LIN {X 0,Y 446.455,Z 877.557,A -85,B 0,C 180,E1 -8817.293,E2 -8817.293} C_VEL
LIN {X 0,Y 446.313,Z 878.965,A -85,B 0,C 180,E1 -8819.098,E2 -8819.098} C_VEL
LIN {X 0,Y 446.282,Z 879.074,A -85,B 0,C 180,E1 -8820,E2 -8820} C_VEL
LIN {X 0,Y 446.28,Z 878.729,A -85,B 0,C 180,E1 -8820.902,E2 -8820.902} C_VEL
LIN {X 0,Y 446.154,Z 876.876,A -85,B 0,C 180,E1 -8822.709,E2 -8822.709} C_VEL
LIN {X 0,Y 446.322,Z 874.333,A -85,B 0,C 180,E1 -8824.063,E2 -8824.063} C_VEL
LIN {X 0,Y 446.471,Z 870.782,A -85,B 0,C 180,E1 -8825.42,E2 -8825.42} C_VEL
LIN {X 0,Y 446.753,Z 866.002,A -85,B 0,C 180,E1 -8826.798,E2 -8826.798} C_VEL
LIN {X 0,Y 446.982,Z 860.13,A -85,B 0,C 180,E1 -8828.135,E2 -8828.135} C_VEL
LIN {X 0,Y 447.259,Z 854.069,A -85,B 0,C 180,E1 -8829.269,E2 -8829.269} C_VEL
LIN {X 0,Y 447.595,Z 846.748,A -85,B 0,C 180,E1 -8830.403,E2 -8830.403} C_VEL
LIN {X 0,Y 447.948,Z 837.847,A -85,B 0,C 180,E1 -8831.539,E2 -8831.539} C_VEL
LIN {X 0,Y 448.295,Z 829.293,A -85,B 0,C 180,E1 -8832.449,E2 -8832.449} C_VEL
LIN {X 0,Y 448.628,Z 820.332,A -85,B 0,C 180,E1 -8833.245,E2 -8833.245} C_VEL
LIN {X 0,Y 448.958,Z 810.568,A -85,B 0,C 180,E1 -8833.959,E2 -8833.959} C_VEL
LIN {X 0,Y 449.192,Z 800.48,A -85,B 0,C 180,E1 -8834.555,E2 -8834.555} C_VEL
LIN {X 0,Y 449.398,Z 790.703,A -85,B 0,C 180,E1 -8835.012,E2 -8835.012} C_VEL
LIN {X 0,Y 449.524,Z 780.049,A -85,B 0,C 180,E1 -8835.385,E2 -8835.385} C_VEL
LIN {X 0,Y 449.624,Z 767.893,A -85,B 0,C 180,E1 -8835.672,E2 -8835.672} C_VEL
LIN {X 0,Y 450.186,Z 707.985,A -85,B 0,C 180,E1 -8836.742,E2 -8836.742} C_VEL
LIN {X 0,Y 446.477,Z 696.872,A -85,B 0,C 180,E1 -8837.1,E2 -8837.1} C_VEL
LIN {X 0,Y 446.458,Z 696.871,A -85,B 0,C 180,E1 -8840.262,E2 -8840.262} C_VEL
LIN {X 0,Y 446.438,Z 696.874,A -85,B 0,C 180,E1 -8843.176,E2 -8843.176} C_VEL
LIN {X 0,Y 446.45,Z 696.87,A -85,B 0,C 180,E1 -8846.19,E2 -8846.19} C_VEL
LIN {X 0,Y 446.452,Z 696.872,A -85,B 0,C 180,E1 -8849.209,E2 -8849.209} C_VEL
LIN {X 0,Y 446.433,Z 696.873,A -85,B 0,C 180,E1 -8852.361,E2 -8852.361} C_VEL
LIN {X 0,Y 446.432,Z 696.871,A -85,B 0,C 180,E1 -8855.625,E2 -8855.625} C_VEL
LIN {X 0,Y 446.424,Z 696.877,A -85,B 0,C 180,E1 -8859.029,E2 -8859.029} C_VEL
LIN {X 0,Y 446.402,Z 696.873,A -85,B 0,C 180,E1 -8862.268,E2 -8862.268} C_VEL
LIN {X 0,Y 446.467,Z 696.872,A -85,B 0,C 180,E1 -8865.102,E2 -8865.102} C_VEL
LIN {X 0,Y 446.417,Z 696.873,A -85,B 0,C 180,E1 -8868.603,E2 -8868.603} C_VEL
LIN {X 0,Y 446.412,Z 696.871,A -85,B 0,C 180,E1 -8871.922,E2 -8871.922} C_VEL
LIN {X 0,Y 446.428,Z 696.874,A -85,B 0,C 180,E1 -8875.472,E2 -8875.472} C_VEL
LIN {X 0,Y 446.404,Z 696.875,A -85,B 0,C 180,E1 -8878.694,E2 -8878.694} C_VEL
LIN {X 0,Y 446.413,Z 696.873,A -85,B 0,C 180,E1 -8881.839,E2 -8881.839} C_VEL
LIN {X 0,Y 446.415,Z 696.876,A -85,B 0,C 180,E1 -8884.84,E2 -8884.84} C_VEL
LIN {X 0,Y 446.457,Z 696.87,A -85,B 0,C 180,E1 -8888.243,E2 -8888.243} C_VEL
LIN {X 0,Y 446.427,Z 696.879,A -85,B 0,C 180,E1 -8891.643,E2 -8891.643} C_VEL
LIN {X 0,Y 446.439,Z 696.875,A -85,B 0,C 180,E1 -8892.562,E2 -8892.562} C_VEL
LIN {X 0,Y 449.167,Z 704.566,A -85,B 0,C 180,E1 -8892.83,E2 -8892.83} C_VEL
LIN {X 0,Y 451.172,Z 709.732,A -85,B 0,C 180,E1 -8892.998,E2 -8892.998} C_VEL
LIN {X 0,Y 451,Z 726.462,A -85,B 0,C 180,E1 -8893.266,E2 -8893.266} C_VEL
LIN {X 0,Y 450.327,Z 732.301,A -85,B 0,C 180,E1 -8893.334,E2 -8893.334} C_VEL
LIN {X 0,Y 444.772,Z 751.316,A -85,B 0,C 180,E1 -8893.421,E2 -8893.421} C_VEL
LIN {X 0,Y 443.989,Z 757.159,A -85,B 0,C 180,E1 -8893.486,E2 -8893.486} C_VEL
LIN {X 0,Y 443.858,Z 779.679,A -85,B 0,C 180,E1 -8893.879,E2 -8893.879} C_VEL
LIN {X 0,Y 443.85,Z 792.762,A -85,B 0,C 180,E1 -8894.291,E2 -8894.291} C_VEL
LIN {X 0,Y 443.58,Z 804.775,A -85,B 0,C 180,E1 -8894.841,E2 -8894.841} C_VEL
LIN {X 0,Y 443.212,Z 816.316,A -85,B 0,C 180,E1 -8895.551,E2 -8895.551} C_VEL
LIN {X 0,Y 442.662,Z 827.625,A -85,B 0,C 180,E1 -8896.451,E2 -8896.451} C_VEL
LIN {X 0,Y 442.145,Z 837.968,A -85,B 0,C 180,E1 -8897.487,E2 -8897.487} C_VEL
LIN {X 0,Y 441.726,Z 846.394,A -85,B 0,C 180,E1 -8898.523,E2 -8898.523} C_VEL
LIN {X 0,Y 441.161,Z 854.165,A -85,B 0,C 180,E1 -8899.67,E2 -8899.67} C_VEL
LIN {X 0,Y 440.632,Z 861.854,A -85,B 0,C 180,E1 -8901.071,E2 -8901.071} C_VEL
LIN {X 0,Y 440.333,Z 867.503,A -85,B 0,C 180,E1 -8902.354,E2 -8902.354} C_VEL
LIN {X 0,Y 439.991,Z 873.273,A -85,B 0,C 180,E1 -8904.035,E2 -8904.035} C_VEL
LIN {X 0,Y 439.577,Z 876.826,A -85,B 0,C 180,E1 -8905.409,E2 -8905.409} C_VEL
LIN {X 0,Y 439.439,Z 878.651,A -85,B 0,C 180,E1 -8906.326,E2 -8906.326} C_VEL
LIN {X 0,Y 439.431,Z 880.017,A -85,B 0,C 180,E1 -8907.244,E2 -8907.244} C_VEL
LIN {X 0,Y 439.368,Z 881.592,A -85,B 0,C 180,E1 -8909.077,E2 -8909.077} C_VEL
LIN {X 0,Y 439.341,Z 881.828,A -85,B 0,C 180,E1 -8909.994,E2 -8909.994} C_VEL
LIN {X 0,Y 439.468,Z 881.071,A -85,B 0,C 180,E1 -8911.827,E2 -8911.827} C_VEL
LIN {X 0,Y 439.428,Z 878.838,A -85,B 0,C 180,E1 -8913.662,E2 -8913.662} C_VEL
LIN {X 0,Y 439.664,Z 876.032,A -85,B 0,C 180,E1 -8915.037,E2 -8915.037} C_VEL
LIN {X 0,Y 440.018,Z 872.218,A -85,B 0,C 180,E1 -8916.413,E2 -8916.413} C_VEL
LIN {X 0,Y 440.314,Z 866.746,A -85,B 0,C 180,E1 -8917.934,E2 -8917.934} C_VEL
LIN {X 0,Y 440.767,Z 859.941,A -85,B 0,C 180,E1 -8919.4,E2 -8919.4} C_VEL
LIN {X 0,Y 441.34,Z 851.927,A -85,B 0,C 180,E1 -8920.777,E2 -8920.777} C_VEL
LIN {X 0,Y 441.868,Z 843.713,A -85,B 0,C 180,E1 -8921.926,E2 -8921.926} C_VEL
LIN {X 0,Y 442.375,Z 833.561,A -85,B 0,C 180,E1 -8923.077,E2 -8923.077} C_VEL
LIN {X 0,Y 442.982,Z 823.11,A -85,B 0,C 180,E1 -8924.024,E2 -8924.024} C_VEL
LIN {X 0,Y 443.404,Z 811.864,A -85,B 0,C 180,E1 -8924.839,E2 -8924.839} C_VEL
LIN {X 0,Y 443.671,Z 800.007,A -85,B 0,C 180,E1 -8925.497,E2 -8925.497} C_VEL
LIN {X 0,Y 443.858,Z 786.655,A -85,B 0,C 180,E1 -8926.02,E2 -8926.02} C_VEL
LIN {X 0,Y 443.867,Z 773.355,A -85,B 0,C 180,E1 -8926.345,E2 -8926.345} C_VEL
LIN {X 0,Y 444.342,Z 711.028,A -85,B 0,C 180,E1 -8927.362,E2 -8927.362} C_VEL
LIN {X 0,Y 439.426,Z 697.751,A -85,B 0,C 180,E1 -8927.803,E2 -8927.803} C_VEL
LIN {X 0,Y 439.371,Z 697.757,A -85,B 0,C 180,E1 -8930.596,E2 -8930.596} C_VEL
LIN {X 0,Y 439.386,Z 697.748,A -85,B 0,C 180,E1 -8934.255,E2 -8934.255} C_VEL
LIN {X 0,Y 439.41,Z 697.746,A -85,B 0,C 180,E1 -8937.626,E2 -8937.626} C_VEL
LIN {X 0,Y 439.331,Z 697.757,A -85,B 0,C 180,E1 -8940.781,E2 -8940.781} C_VEL
LIN {X 0,Y 439.354,Z 697.753,A -85,B 0,C 180,E1 -8944.037,E2 -8944.037} C_VEL
LIN {X 0,Y 439.324,Z 697.755,A -85,B 0,C 180,E1 -8947.427,E2 -8947.427} C_VEL
LIN {X 0,Y 439.386,Z 697.755,A -85,B 0,C 180,E1 -8949.846,E2 -8949.846} C_VEL
LIN {X 0,Y 439.359,Z 697.754,A -85,B 0,C 180,E1 -8952.623,E2 -8952.623} C_VEL
LIN {X 0,Y 439.355,Z 697.751,A -85,B 0,C 180,E1 -8956.027,E2 -8956.027} C_VEL
LIN {X 0,Y 439.35,Z 697.756,A -85,B 0,C 180,E1 -8959.015,E2 -8959.015} C_VEL
LIN {X 0,Y 439.341,Z 697.757,A -85,B 0,C 180,E1 -8961.598,E2 -8961.598} C_VEL
LIN {X 0,Y 439.343,Z 697.753,A -85,B 0,C 180,E1 -8964.839,E2 -8964.839} C_VEL
LIN {X 0,Y 439.328,Z 697.763,A -85,B 0,C 180,E1 -8968.136,E2 -8968.136} C_VEL
LIN {X 0,Y 439.362,Z 697.746,A -85,B 0,C 180,E1 -8971.322,E2 -8971.322} C_VEL
LIN {X 0,Y 439.347,Z 697.757,A -85,B 0,C 180,E1 -8974.411,E2 -8974.411} C_VEL
LIN {X 0,Y 439.297,Z 697.756,A -85,B 0,C 180,E1 -8977.421,E2 -8977.421} C_VEL
LIN {X 0,Y 439.371,Z 697.753,A -85,B 0,C 180,E1 -8980.66,E2 -8980.66} C_VEL
LIN {X 0,Y 439.405,Z 697.746,A -85,B 0,C 180,E1 -8984.222,E2 -8984.222} C_VEL
LIN {X 0,Y 439.44,Z 697.742,A -85,B 0,C 180,E1 -8988,E2 -8988} C_VEL
LIN {X 0,Y 439.474,Z 697.739,A -85,B 0,C 180,E1 -8991.725,E2 -8991.725} C_VEL
LIN {X 0,Y 439.553,Z 697.733,A -85,B 0,C 180,E1 -8994.495,E2 -8994.495} C_VEL
LIN {X 0,Y 439.591,Z 697.728,A -85,B 0,C 180,E1 -8997.251,E2 -8997.251} C_VEL
LIN {X 0,Y 439.687,Z 697.714,A -85,B 0,C 180,E1 -9000,E2 -9000} C_VEL
LIN {X 0,Y 439.591,Z 697.724,A -85,B 0,C 180,E1 -9002.749,E2 -9002.749} C_VEL
LIN {X 0,Y 439.546,Z 697.731,A -85,B 0,C 180,E1 -9006.426,E2 -9006.426} C_VEL
LIN {X 0,Y 439.431,Z 697.744,A -85,B 0,C 180,E1 -9009.203,E2 -9009.203} C_VEL
LIN {X 0,Y 439.431,Z 697.745,A -85,B 0,C 180,E1 -9012.729,E2 -9012.729} C_VEL
LIN {X 0,Y 439.388,Z 697.748,A -85,B 0,C 180,E1 -9016.357,E2 -9016.357} C_VEL
LIN {X 0,Y 439.332,Z 697.758,A -85,B 0,C 180,E1 -9019.63,E2 -9019.63} C_VEL
LIN {X 0,Y 439.299,Z 697.759,A -85,B 0,C 180,E1 -9022.579,E2 -9022.579} C_VEL
LIN {X 0,Y 439.348,Z 697.755,A -85,B 0,C 180,E1 -9025.588,E2 -9025.588} C_VEL
LIN {X 0,Y 439.361,Z 697.751,A -85,B 0,C 180,E1 -9028.678,E2 -9028.678} C_VEL
LIN {X 0,Y 439.323,Z 697.764,A -85,B 0,C 180,E1 -9032.038,E2 -9032.038} C_VEL
LIN {X 0,Y 439.338,Z 697.755,A -85,B 0,C 180,E1 -9035.346,E2 -9035.346} C_VEL
LIN {X 0,Y 439.347,Z 697.747,A -85,B 0,C 180,E1 -9038.599,E2 -9038.599} C_VEL
LIN {X 0,Y 439.354,Z 697.754,A -85,B 0,C 180,E1 -9041.265,E2 -9041.265} C_VEL
LIN {X 0,Y 439.362,Z 697.756,A -85,B 0,C 180,E1 -9044.735,E2 -9044.735} C_VEL
LIN {X 0,Y 439.368,Z 697.749,A -85,B 0,C 180,E1 -9047.804,E2 -9047.804} C_VEL
LIN {X 0,Y 439.409,Z 697.751,A -85,B 0,C 180,E1 -9050.237,E2 -9050.237} C_VEL
LIN {X 0,Y 439.339,Z 697.756,A -85,B 0,C 180,E1 -9053.72,E2 -9053.72} C_VEL
LIN {X 0,Y 439.339,Z 697.752,A -85,B 0,C 180,E1 -9057.061,E2 -9057.061} C_VEL
LIN {X 0,Y 439.372,Z 697.924,A -85,B 0,C 180,E1 -9058.351,E2 -9058.351} C_VEL
LIN {X 0,Y 442.863,Z 712.769,A -85,B 0,C 180,E1 -9060.789,E2 -9060.789} C_VEL
LIN {X 0,Y 444.145,Z 719.99,A -85,B 0,C 180,E1 -9061.916,E2 -9061.916} C_VEL
LIN {X 0,Y 443.017,Z 740.571,A -85,B 0,C 180,E1 -9064.839,E2 -9064.839} C_VEL
LIN {X 0,Y 441.856,Z 763.5,A -85,B 0,C 180,E1 -9068.059,E2 -9068.059} C_VEL
LIN {X 0,Y 440.667,Z 790.642,A -85,B 0,C 180,E1 -9071.854,E2 -9071.854} C_VEL
LIN {X 0,Y 443.804,Z 820.24,A -85,B 0,C 180,E1 -9072.469,E2 -9072.469} C_VEL
LIN {X 0,Y 443.016,Z 901.258,A -85,B 0,C 180,E1 -9073.801,E2 -9073.801} C_VEL
LIN {X 0,Y 442.55,Z 914.493,A -85,B 0,C 180,E1 -9074.197,E2 -9074.197} C_VEL
LIN {X 0,Y 441.94,Z 926.688,A -85,B 0,C 180,E1 -9074.736,E2 -9074.736} C_VEL
LIN {X 0,Y 441.232,Z 939.047,A -85,B 0,C 180,E1 -9075.478,E2 -9075.478} C_VEL
LIN {X 0,Y 440.652,Z 950.666,A -85,B 0,C 180,E1 -9076.391,E2 -9076.391} C_VEL
LIN {X 0,Y 440.182,Z 961.387,A -85,B 0,C 180,E1 -9077.443,E2 -9077.443} C_VEL
LIN {X 0,Y 439.599,Z 970.058,A -85,B 0,C 180,E1 -9078.479,E2 -9078.479} C_VEL
LIN {X 0,Y 439.2,Z 978.094,A -85,B 0,C 180,E1 -9079.636,E2 -9079.636} C_VEL
LIN {X 0,Y 438.891,Z 985.975,A -85,B 0,C 180,E1 -9081.025,E2 -9081.025} C_VEL
LIN {X 0,Y 438.757,Z 991.39,A -85,B 0,C 180,E1 -9082.181,E2 -9082.181} C_VEL
LIN {X 0,Y 438.677,Z 996.651,A -85,B 0,C 180,E1 -9083.568,E2 -9083.568} C_VEL
LIN {X 0,Y 438.691,Z 1000.753,A -85,B 0,C 180,E1 -9084.951,E2 -9084.951} C_VEL
LIN {X 0,Y 438.734,Z 1003.79,A -85,B 0,C 180,E1 -9086.333,E2 -9086.333} C_VEL
LIN {X 0,Y 438.697,Z 1005.225,A -85,B 0,C 180,E1 -9087.252,E2 -9087.252} C_VEL
LIN {X 0,Y 438.702,Z 1006.253,A -85,B 0,C 180,E1 -9088.17,E2 -9088.17} C_VEL
LIN {X 0,Y 438.698,Z 1006.878,A -85,B 0,C 180,E1 -9089.088,E2 -9089.088} C_VEL
LIN {X 0,Y 438.706,Z 1007.099,A -85,B 0,C 180,E1 -9090.006,E2 -9090.006} C_VEL
LIN {X 0,Y 438.699,Z 1006.871,A -85,B 0,C 180,E1 -9090.924,E2 -9090.924} C_VEL
LIN {X 0,Y 438.703,Z 1006.24,A -85,B 0,C 180,E1 -9091.842,E2 -9091.842} C_VEL
LIN {X 0,Y 438.699,Z 1005.207,A -85,B 0,C 180,E1 -9092.761,E2 -9092.761} C_VEL
LIN {X 0,Y 438.738,Z 1003.764,A -85,B 0,C 180,E1 -9093.68,E2 -9093.68} C_VEL
LIN {X 0,Y 438.697,Z 1000.723,A -85,B 0,C 180,E1 -9095.061,E2 -9095.061} C_VEL
LIN {X 0,Y 438.691,Z 995.886,A -85,B 0,C 180,E1 -9096.652,E2 -9096.652} C_VEL
LIN {X 0,Y 438.806,Z 989.268,A -85,B 0,C 180,E1 -9098.293,E2 -9098.293} C_VEL
LIN {X 0,Y 439.038,Z 982.182,A -85,B 0,C 180,E1 -9099.682,E2 -9099.682} C_VEL
LIN {X 0,Y 439.436,Z 973.342,A -85,B 0,C 180,E1 -9101.07,E2 -9101.07} C_VEL
LIN {X 0,Y 439.934,Z 964.317,A -85,B 0,C 180,E1 -9102.226,E2 -9102.226} C_VEL
LIN {X 0,Y 440.416,Z 954.695,A -85,B 0,C 180,E1 -9103.24,E2 -9103.24} C_VEL
LIN {X 0,Y 440.988,Z 943.632,A -85,B 0,C 180,E1 -9104.189,E2 -9104.189} C_VEL
LIN {X 0,Y 441.695,Z 931.622,A -85,B 0,C 180,E1 -9104.99,E2 -9104.99} C_VEL
LIN {X 0,Y 442.316,Z 919.158,A -85,B 0,C 180,E1 -9105.617,E2 -9105.617} C_VEL
LIN {X 0,Y 442.865,Z 906.362,A -85,B 0,C 180,E1 -9106.07,E2 -9106.07} C_VEL
LIN {X 0,Y 443.13,Z 892.903,A -85,B 0,C 180,E1 -9106.356,E2 -9106.356} C_VEL
LIN {X 0,Y 443.769,Z 818.643,A -85,B 0,C 180,E1 -9107.557,E2 -9107.557} C_VEL
LIN {X 0,Y 440.666,Z 790.416,A -85,B 0,C 180,E1 -9108.15,E2 -9108.15} C_VEL
LIN {X 0,Y 441.837,Z 763.389,A -85,B 0,C 180,E1 -9111.955,E2 -9111.955} C_VEL
LIN {X 0,Y 443.087,Z 739.566,A -85,B 0,C 180,E1 -9115.297,E2 -9115.297} C_VEL
LIN {X 0,Y 444.132,Z 719.77,A -85,B 0,C 180,E1 -9118.113,E2 -9118.113} C_VEL
LIN {X 0,Y 441.965,Z 709.09,A -85,B 0,C 180,E1 -9119.802,E2 -9119.802} C_VEL
LIN {X 0,Y 439.36,Z 697.755,A -85,B 0,C 180,E1 -9121.698,E2 -9121.698} C_VEL
LIN {X 0,Y 439.347,Z 697.751,A -85,B 0,C 180,E1 -9125.165,E2 -9125.165} C_VEL
LIN {X 0,Y 439.361,Z 697.756,A -85,B 0,C 180,E1 -9128.602,E2 -9128.602} C_VEL
LIN {X 0,Y 439.36,Z 697.753,A -85,B 0,C 180,E1 -9132.213,E2 -9132.213} C_VEL
LIN {X 0,Y 439.386,Z 697.756,A -85,B 0,C 180,E1 -9135.269,E2 -9135.269} C_VEL
LIN {X 0,Y 439.379,Z 697.752,A -85,B 0,C 180,E1 -9138.749,E2 -9138.749} C_VEL
LIN {X 0,Y 439.373,Z 697.755,A -85,B 0,C 180,E1 -9141.613,E2 -9141.613} C_VEL
LIN {X 0,Y 439.409,Z 697.749,A -85,B 0,C 180,E1 -9144.845,E2 -9144.845} C_VEL
LIN {X 0,Y 439.387,Z 697.75,A -85,B 0,C 180,E1 -9148.141,E2 -9148.141} C_VEL
LIN {X 0,Y 439.418,Z 697.75,A -85,B 0,C 180,E1 -9151.607,E2 -9151.607} C_VEL
LIN {X 0,Y 439.391,Z 697.752,A -85,B 0,C 180,E1 -9154.414,E2 -9154.414} C_VEL
LIN {X 0,Y 439.378,Z 697.756,A -85,B 0,C 180,E1 -9157.425,E2 -9157.425} C_VEL
LIN {X 0,Y 439.457,Z 697.746,A -85,B 0,C 180,E1 -9160.664,E2 -9160.664} C_VEL
LIN {X 0,Y 439.439,Z 697.748,A -85,B 0,C 180,E1 -9162.235,E2 -9162.235} C_VEL
LIN {X 0,Y 441.356,Z 702.841,A -85,B 0,C 180,E1 -9162.452,E2 -9162.452} C_VEL
LIN {X 0,Y 444.315,Z 710.253,A -85,B 0,C 180,E1 -9162.766,E2 -9162.766} C_VEL
LIN {X 0,Y 443.368,Z 779.682,A -85,B 0,C 180,E1 -9164.161,E2 -9164.161} C_VEL
LIN {X 0,Y 443.253,Z 791.804,A -85,B 0,C 180,E1 -9164.54,E2 -9164.54} C_VEL
LIN {X 0,Y 443.078,Z 802.332,A -85,B 0,C 180,E1 -9165.004,E2 -9165.004} C_VEL
LIN {X 0,Y 442.813,Z 812.088,A -85,B 0,C 180,E1 -9165.56,E2 -9165.56} C_VEL
LIN {X 0,Y 442.508,Z 821.385,A -85,B 0,C 180,E1 -9166.218,E2 -9166.218} C_VEL
LIN {X 0,Y 442.072,Z 830.698,A -85,B 0,C 180,E1 -9167.023,E2 -9167.023} C_VEL
LIN {X 0,Y 441.757,Z 838.477,A -85,B 0,C 180,E1 -9167.831,E2 -9167.831} C_VEL
LIN {X 0,Y 441.36,Z 845.982,A -85,B 0,C 180,E1 -9168.752,E2 -9168.752} C_VEL
LIN {X 0,Y 440.902,Z 853.731,A -85,B 0,C 180,E1 -9169.902,E2 -9169.902} C_VEL
LIN {X 0,Y 440.565,Z 860.129,A -85,B 0,C 180,E1 -9171.052,E2 -9171.052} C_VEL
LIN {X 0,Y 440.223,Z 866.217,A -85,B 0,C 180,E1 -9172.397,E2 -9172.397} C_VEL
LIN {X 0,Y 439.932,Z 870.545,A -85,B 0,C 180,E1 -9173.579,E2 -9173.579} C_VEL
LIN {X 0,Y 439.654,Z 873.382,A -85,B 0,C 180,E1 -9174.496,E2 -9174.496} C_VEL
LIN {X 0,Y 439.482,Z 877.281,A -85,B 0,C 180,E1 -9176.333,E2 -9176.333} C_VEL
LIN {X 0,Y 439.465,Z 878.682,A -85,B 0,C 180,E1 -9177.25,E2 -9177.25} C_VEL
LIN {X 0,Y 439.299,Z 880.057,A -85,B 0,C 180,E1 -9179.083,E2 -9179.083} C_VEL
LIN {X 0,Y 439.267,Z 880.138,A -85,B 0,C 180,E1 -9180,E2 -9180} C_VEL
LIN {X 0,Y 439.266,Z 879.765,A -85,B 0,C 180,E1 -9180.917,E2 -9180.917} C_VEL
LIN {X 0,Y 439.131,Z 877.857,A -85,B 0,C 180,E1 -9182.752,E2 -9182.752} C_VEL
LIN {X 0,Y 439.304,Z 875.263,A -85,B 0,C 180,E1 -9184.128,E2 -9184.128} C_VEL
LIN {X 0,Y 439.473,Z 871.652,A -85,B 0,C 180,E1 -9185.506,E2 -9185.506} C_VEL
LIN {X 0,Y 439.758,Z 866.895,A -85,B 0,C 180,E1 -9186.884,E2 -9186.884} C_VEL
LIN {X 0,Y 439.993,Z 860.846,A -85,B 0,C 180,E1 -9188.265,E2 -9188.265} C_VEL
LIN {X 0,Y 440.299,Z 854.707,A -85,B 0,C 180,E1 -9189.417,E2 -9189.417} C_VEL
LIN {X 0,Y 440.635,Z 847.294,A -85,B 0,C 180,E1 -9190.569,E2 -9190.569} C_VEL
LIN {X 0,Y 440.949,Z 839.299,A -85,B 0,C 180,E1 -9191.608,E2 -9191.608} C_VEL
LIN {X 0,Y 441.346,Z 830.818,A -85,B 0,C 180,E1 -9192.531,E2 -9192.531} C_VEL
LIN {X 0,Y 441.677,Z 821.96,A -85,B 0,C 180,E1 -9193.34,E2 -9193.34} C_VEL
LIN {X 0,Y 442.013,Z 812.037,A -85,B 0,C 180,E1 -9194.085,E2 -9194.085} C_VEL
LIN {X 0,Y 442.263,Z 801.34,A -85,B 0,C 180,E1 -9194.73,E2 -9194.73} C_VEL
LIN {X 0,Y 442.494,Z 791.555,A -85,B 0,C 180,E1 -9195.193,E2 -9195.193} C_VEL
LIN {X 0,Y 442.623,Z 780.909,A -85,B 0,C 180,E1 -9195.572,E2 -9195.572} C_VEL
LIN {X 0,Y 442.722,Z 768.843,A -85,B 0,C 180,E1 -9195.863,E2 -9195.863} C_VEL
LIN {X 0,Y 443.311,Z 709.347,A -85,B 0,C 180,E1 -9196.955,E2 -9196.955} C_VEL
LIN {X 0,Y 439.451,Z 697.745,A -85,B 0,C 180,E1 -9197.315,E2 -9197.315} C_VEL
LIN {X 0,Y 439.418,Z 697.746,A -85,B 0,C 180,E1 -9199.626,E2 -9199.626} C_VEL
LIN {X 0,Y 439.377,Z 697.754,A -85,B 0,C 180,E1 -9202.575,E2 -9202.575} C_VEL
LIN {X 0,Y 439.392,Z 697.749,A -85,B 0,C 180,E1 -9205.586,E2 -9205.586} C_VEL
LIN {X 0,Y 439.413,Z 697.75,A -85,B 0,C 180,E1 -9208.674,E2 -9208.674} C_VEL
LIN {X 0,Y 439.382,Z 697.75,A -85,B 0,C 180,E1 -9212.028,E2 -9212.028} C_VEL
LIN {X 0,Y 439.407,Z 697.748,A -85,B 0,C 180,E1 -9215.338,E2 -9215.338} C_VEL
LIN {X 0,Y 439.379,Z 697.752,A -85,B 0,C 180,E1 -9218.596,E2 -9218.596} C_VEL
LIN {X 0,Y 439.369,Z 697.749,A -85,B 0,C 180,E1 -9222.208,E2 -9222.208} C_VEL
LIN {X 0,Y 439.414,Z 697.748,A -85,B 0,C 180,E1 -9225.268,E2 -9225.268} C_VEL
LIN {X 0,Y 439.37,Z 697.754,A -85,B 0,C 180,E1 -9229.014,E2 -9229.014} C_VEL
LIN {X 0,Y 439.372,Z 697.75,A -85,B 0,C 180,E1 -9231.609,E2 -9231.609} C_VEL
LIN {X 0,Y 439.403,Z 697.748,A -85,B 0,C 180,E1 -9234.84,E2 -9234.84} C_VEL
LIN {X 0,Y 439.361,Z 697.75,A -85,B 0,C 180,E1 -9238.134,E2 -9238.134} C_VEL
LIN {X 0,Y 439.392,Z 697.754,A -85,B 0,C 180,E1 -9241.32,E2 -9241.32} C_VEL
LIN {X 0,Y 439.354,Z 697.753,A -85,B 0,C 180,E1 -9244.407,E2 -9244.407} C_VEL
LIN {X 0,Y 439.364,Z 697.759,A -85,B 0,C 180,E1 -9247.42,E2 -9247.42} C_VEL
LIN {X 0,Y 439.394,Z 697.752,A -85,B 0,C 180,E1 -9250.682,E2 -9250.682} C_VEL
LIN {X 0,Y 439.433,Z 697.748,A -85,B 0,C 180,E1 -9252.289,E2 -9252.289} C_VEL
LIN {X 0,Y 444.398,Z 711.275,A -85,B 0,C 180,E1 -9252.74,E2 -9252.74} C_VEL
LIN {X 0,Y 443.989,Z 757.159,A -85,B 0,C 180,E1 -9253.486,E2 -9253.486} C_VEL
LIN {X 0,Y 443.229,Z 763.002,A -85,B 0,C 180,E1 -9253.548,E2 -9253.548} C_VEL
LIN {X 0,Y 437.823,Z 781.983,A -85,B 0,C 180,E1 -9253.685,E2 -9253.685} C_VEL
LIN {X 0,Y 437.147,Z 787.717,A -85,B 0,C 180,E1 -9253.825,E2 -9253.825} C_VEL
LIN {X 0,Y 436.944,Z 799.963,A -85,B 0,C 180,E1 -9254.306,E2 -9254.306} C_VEL
LIN {X 0,Y 436.572,Z 812.007,A -85,B 0,C 180,E1 -9254.962,E2 -9254.962} C_VEL
LIN {X 0,Y 436.141,Z 823.948,A -85,B 0,C 180,E1 -9255.833,E2 -9255.833} C_VEL
LIN {X 0,Y 435.534,Z 834.659,A -85,B 0,C 180,E1 -9256.82,E2 -9256.82} C_VEL
LIN {X 0,Y 435.024,Z 843.868,A -85,B 0,C 180,E1 -9257.871,E2 -9257.871} C_VEL
LIN {X 0,Y 434.471,Z 852.258,A -85,B 0,C 180,E1 -9259.038,E2 -9259.038} C_VEL
LIN {X 0,Y 433.851,Z 860.393,A -85,B 0,C 180,E1 -9260.437,E2 -9260.437} C_VEL
LIN {X 0,Y 433.373,Z 867.275,A -85,B 0,C 180,E1 -9261.92,E2 -9261.92} C_VEL
LIN {X 0,Y 433.069,Z 872.895,A -85,B 0,C 180,E1 -9263.471,E2 -9263.471} C_VEL
LIN {X 0,Y 432.672,Z 876.788,A -85,B 0,C 180,E1 -9264.869,E2 -9264.869} C_VEL
LIN {X 0,Y 432.425,Z 879.655,A -85,B 0,C 180,E1 -9266.267,E2 -9266.267} C_VEL
LIN {X 0,Y 432.414,Z 881.019,A -85,B 0,C 180,E1 -9267.199,E2 -9267.199} C_VEL
LIN {X 0,Y 432.348,Z 882.594,A -85,B 0,C 180,E1 -9269.062,E2 -9269.062} C_VEL
LIN {X 0,Y 432.318,Z 882.83,A -85,B 0,C 180,E1 -9269.994,E2 -9269.994} C_VEL
LIN {X 0,Y 432.449,Z 882.072,A -85,B 0,C 180,E1 -9271.856,E2 -9271.856} C_VEL
LIN {X 0,Y 432.414,Z 879.84,A -85,B 0,C 180,E1 -9273.721,E2 -9273.721} C_VEL
LIN {X 0,Y 432.664,Z 877.033,A -85,B 0,C 180,E1 -9275.119,E2 -9275.119} C_VEL
LIN {X 0,Y 433.04,Z 873.218,A -85,B 0,C 180,E1 -9276.517,E2 -9276.517} C_VEL
LIN {X 0,Y 433.355,Z 867.746,A -85,B 0,C 180,E1 -9278.062,E2 -9278.062} C_VEL
LIN {X 0,Y 433.835,Z 860.941,A -85,B 0,C 180,E1 -9279.551,E2 -9279.551} C_VEL
LIN {X 0,Y 434.441,Z 852.926,A -85,B 0,C 180,E1 -9280.95,E2 -9280.95} C_VEL
LIN {X 0,Y 434.994,Z 844.712,A -85,B 0,C 180,E1 -9282.117,E2 -9282.117} C_VEL
LIN {X 0,Y 435.532,Z 834.559,A -85,B 0,C 180,E1 -9283.287,E2 -9283.287} C_VEL
LIN {X 0,Y 436.167,Z 824.107,A -85,B 0,C 180,E1 -9284.248,E2 -9284.248} C_VEL
LIN {X 0,Y 436.613,Z 812.86,A -85,B 0,C 180,E1 -9285.075,E2 -9285.075} C_VEL
LIN {X 0,Y 436.918,Z 800.997,A -85,B 0,C 180,E1 -9285.742,E2 -9285.742} C_VEL
LIN {X 0,Y 437.089,Z 787.647,A -85,B 0,C 180,E1 -9286.275,E2 -9286.275} C_VEL
LIN {X 0,Y 437.095,Z 774.335,A -85,B 0,C 180,E1 -9286.605,E2 -9286.605} C_VEL
LIN {X 0,Y 437.584,Z 712.545,A -85,B 0,C 180,E1 -9287.63,E2 -9287.63} C_VEL
LIN {X 0,Y 432.385,Z 698.628,A -85,B 0,C 180,E1 -9288.103,E2 -9288.103} C_VEL
LIN {X 0,Y 432.332,Z 698.634,A -85,B 0,C 180,E1 -9290.947,E2 -9290.947} C_VEL
LIN {X 0,Y 432.354,Z 698.625,A -85,B 0,C 180,E1 -9294.454,E2 -9294.454} C_VEL
LIN {X 0,Y 432.36,Z 698.628,A -85,B 0,C 180,E1 -9297.065,E2 -9297.065} C_VEL
LIN {X 0,Y 432.318,Z 698.629,A -85,B 0,C 180,E1 -9300.503,E2 -9300.503} C_VEL
LIN {X 0,Y 432.326,Z 698.628,A -85,B 0,C 180,E1 -9303.996,E2 -9303.996} C_VEL
LIN {X 0,Y 432.295,Z 698.635,A -85,B 0,C 180,E1 -9307.192,E2 -9307.192} C_VEL
LIN {X 0,Y 432.316,Z 698.633,A -85,B 0,C 180,E1 -9310.176,E2 -9310.176} C_VEL
LIN {X 0,Y 432.321,Z 698.633,A -85,B 0,C 180,E1 -9313.048,E2 -9313.048} C_VEL
LIN {X 0,Y 432.331,Z 698.621,A -85,B 0,C 180,E1 -9315.652,E2 -9315.652} C_VEL
LIN {X 0,Y 432.323,Z 698.632,A -85,B 0,C 180,E1 -9318.386,E2 -9318.386} C_VEL
LIN {X 0,Y 432.3,Z 698.635,A -85,B 0,C 180,E1 -9321.846,E2 -9321.846} C_VEL
LIN {X 0,Y 432.283,Z 698.633,A -85,B 0,C 180,E1 -9325.317,E2 -9325.317} C_VEL
LIN {X 0,Y 432.272,Z 698.636,A -85,B 0,C 180,E1 -9328.65,E2 -9328.65} C_VEL
LIN {X 0,Y 432.321,Z 698.627,A -85,B 0,C 180,E1 -9331.872,E2 -9331.872} C_VEL
LIN {X 0,Y 432.291,Z 698.631,A -85,B 0,C 180,E1 -9334.995,E2 -9334.995} C_VEL
LIN {X 0,Y 432.289,Z 698.633,A -85,B 0,C 180,E1 -9338.042,E2 -9338.042} C_VEL
LIN {X 0,Y 432.315,Z 698.628,A -85,B 0,C 180,E1 -9341.026,E2 -9341.026} C_VEL
LIN {X 0,Y 432.372,Z 698.62,A -85,B 0,C 180,E1 -9343.959,E2 -9343.959} C_VEL
LIN {X 0,Y 432.411,Z 698.617,A -85,B 0,C 180,E1 -9347.802,E2 -9347.802} C_VEL
LIN {X 0,Y 432.419,Z 698.618,A -85,B 0,C 180,E1 -9351.589,E2 -9351.589} C_VEL
LIN {X 0,Y 432.528,Z 698.607,A -85,B 0,C 180,E1 -9354.405,E2 -9354.405} C_VEL
LIN {X 0,Y 432.532,Z 698.604,A -85,B 0,C 180,E1 -9358.138,E2 -9358.138} C_VEL
LIN {X 0,Y 432.658,Z 698.589,A -85,B 0,C 180,E1 -9360,E2 -9360} C_VEL
LIN {X 0,Y 432.541,Z 698.602,A -85,B 0,C 180,E1 -9362.794,E2 -9362.794} C_VEL
LIN {X 0,Y 432.5,Z 698.61,A -85,B 0,C 180,E1 -9366.531,E2 -9366.531} C_VEL
LIN {X 0,Y 432.375,Z 698.623,A -85,B 0,C 180,E1 -9369.355,E2 -9369.355} C_VEL
LIN {X 0,Y 432.372,Z 698.625,A -85,B 0,C 180,E1 -9372.814,E2 -9372.814} C_VEL
LIN {X 0,Y 432.351,Z 698.624,A -85,B 0,C 180,E1 -9376.486,E2 -9376.486} C_VEL
LIN {X 0,Y 432.268,Z 698.633,A -85,B 0,C 180,E1 -9379.964,E2 -9379.964} C_VEL
LIN {X 0,Y 432.254,Z 698.637,A -85,B 0,C 180,E1 -9382.968,E2 -9382.968} C_VEL
LIN {X 0,Y 432.303,Z 698.631,A -85,B 0,C 180,E1 -9386.036,E2 -9386.036} C_VEL
LIN {X 0,Y 432.289,Z 698.633,A -85,B 0,C 180,E1 -9389.191,E2 -9389.191} C_VEL
LIN {X 0,Y 432.272,Z 698.638,A -85,B 0,C 180,E1 -9392.3,E2 -9392.3} C_VEL
LIN {X 0,Y 432.282,Z 698.634,A -85,B 0,C 180,E1 -9394.682,E2 -9394.682} C_VEL
LIN {X 0,Y 432.3,Z 698.627,A -85,B 0,C 180,E1 -9398.154,E2 -9398.154} C_VEL
LIN {X 0,Y 432.322,Z 698.631,A -85,B 0,C 180,E1 -9401.614,E2 -9401.614} C_VEL
LIN {X 0,Y 432.331,Z 698.634,A -85,B 0,C 180,E1 -9404.348,E2 -9404.348} C_VEL
LIN {X 0,Y 432.321,Z 698.626,A -85,B 0,C 180,E1 -9407.016,E2 -9407.016} C_VEL
LIN {X 0,Y 432.316,Z 698.633,A -85,B 0,C 180,E1 -9409.824,E2 -9409.824} C_VEL
LIN {X 0,Y 432.278,Z 698.636,A -85,B 0,C 180,E1 -9413.03,E2 -9413.03} C_VEL
LIN {X 0,Y 432.325,Z 698.622,A -85,B 0,C 180,E1 -9416.004,E2 -9416.004} C_VEL
LIN {X 0,Y 432.316,Z 698.708,A -85,B 0,C 180,E1 -9418.041,E2 -9418.041} C_VEL
LIN {X 0,Y 436.106,Z 714.882,A -85,B 0,C 180,E1 -9420.747,E2 -9420.747} C_VEL
LIN {X 0,Y 437.239,Z 720.888,A -85,B 0,C 180,E1 -9421.704,E2 -9421.704} C_VEL
LIN {X 0,Y 436.121,Z 740.883,A -85,B 0,C 180,E1 -9424.597,E2 -9424.597} C_VEL
LIN {X 0,Y 434.988,Z 762.527,A -85,B 0,C 180,E1 -9427.694,E2 -9427.694} C_VEL
LIN {X 0,Y 433.691,Z 789.692,A -85,B 0,C 180,E1 -9431.553,E2 -9431.553} C_VEL
LIN {X 0,Y 437.023,Z 820.942,A -85,B 0,C 180,E1 -9432.217,E2 -9432.217} C_VEL
LIN {X 0,Y 436.21,Z 900.257,A -85,B 0,C 180,E1 -9433.541,E2 -9433.541} C_VEL
LIN {X 0,Y 435.684,Z 913.482,A -85,B 0,C 180,E1 -9433.941,E2 -9433.941} C_VEL
LIN {X 0,Y 435.03,Z 925.671,A -85,B 0,C 180,E1 -9434.488,E2 -9434.488} C_VEL
LIN {X 0,Y 434.294,Z 938.028,A -85,B 0,C 180,E1 -9435.241,E2 -9435.241} C_VEL
LIN {X 0,Y 433.694,Z 949.747,A -85,B 0,C 180,E1 -9436.177,E2 -9436.177} C_VEL
LIN {X 0,Y 433.224,Z 959.275,A -85,B 0,C 180,E1 -9437.118,E2 -9437.118} C_VEL
LIN {X 0,Y 432.562,Z 969.035,A -85,B 0,C 180,E1 -9438.289,E2 -9438.289} C_VEL
LIN {X 0,Y 432.162,Z 977.075,A -85,B 0,C 180,E1 -9439.465,E2 -9439.465} C_VEL
LIN {X 0,Y 431.839,Z 984.957,A -85,B 0,C 180,E1 -9440.877,E2 -9440.877} C_VEL
LIN {X 0,Y 431.677,Z 992.25,A -85,B 0,C 180,E1 -9442.523,E2 -9442.523} C_VEL
LIN {X 0,Y 431.638,Z 997.12,A -85,B 0,C 180,E1 -9443.931,E2 -9443.931} C_VEL
LIN {X 0,Y 431.663,Z 1000.855,A -85,B 0,C 180,E1 -9445.337,E2 -9445.337} C_VEL
LIN {X 0,Y 431.697,Z 1002.784,A -85,B 0,C 180,E1 -9446.273,E2 -9446.273} C_VEL
LIN {X 0,Y 431.656,Z 1004.22,A -85,B 0,C 180,E1 -9447.207,E2 -9447.207} C_VEL
LIN {X 0,Y 431.665,Z 1005.249,A -85,B 0,C 180,E1 -9448.14,E2 -9448.14} C_VEL
LIN {X 0,Y 431.667,Z 1005.875,A -85,B 0,C 180,E1 -9449.073,E2 -9449.073} C_VEL
LIN {X 0,Y 431.677,Z 1006.096,A -85,B 0,C 180,E1 -9450.006,E2 -9450.006} C_VEL
LIN {X 0,Y 431.667,Z 1005.868,A -85,B 0,C 180,E1 -9450.939,E2 -9450.939} C_VEL
LIN {X 0,Y 431.665,Z 1005.236,A -85,B 0,C 180,E1 -9451.872,E2 -9451.872} C_VEL
LIN {X 0,Y 431.658,Z 1004.201,A -85,B 0,C 180,E1 -9452.806,E2 -9452.806} C_VEL
LIN {X 0,Y 431.701,Z 1002.758,A -85,B 0,C 180,E1 -9453.74,E2 -9453.74} C_VEL
LIN {X 0,Y 431.637,Z 999.711,A -85,B 0,C 180,E1 -9455.144,E2 -9455.144} C_VEL
LIN {X 0,Y 431.618,Z 995.246,A -85,B 0,C 180,E1 -9456.656,E2 -9456.656} C_VEL
LIN {X 0,Y 431.719,Z 989.289,A -85,B 0,C 180,E1 -9458.195,E2 -9458.195} C_VEL
LIN {X 0,Y 431.928,Z 982.425,A -85,B 0,C 180,E1 -9459.606,E2 -9459.606} C_VEL
LIN {X 0,Y 432.335,Z 973.948,A -85,B 0,C 180,E1 -9461.017,E2 -9461.017} C_VEL
LIN {X 0,Y 432.794,Z 965.274,A -85,B 0,C 180,E1 -9462.192,E2 -9462.192} C_VEL
LIN {X 0,Y 433.379,Z 954.836,A -85,B 0,C 180,E1 -9463.342,E2 -9463.342} C_VEL
LIN {X 0,Y 433.963,Z 944.055,A -85,B 0,C 180,E1 -9464.304,E2 -9464.304} C_VEL
LIN {X 0,Y 434.674,Z 932.551,A -85,B 0,C 180,E1 -9465.118,E2 -9465.118} C_VEL
LIN {X 0,Y 435.327,Z 920.752,A -85,B 0,C 180,E1 -9465.754,E2 -9465.754} C_VEL
LIN {X 0,Y 435.977,Z 907.186,A -85,B 0,C 180,E1 -9466.271,E2 -9466.271} C_VEL
LIN {X 0,Y 436.296,Z 893.668,A -85,B 0,C 180,E1 -9466.589,E2 -9466.589} C_VEL
LIN {X 0,Y 436.96,Z 819.227,A -85,B 0,C 180,E1 -9467.813,E2 -9467.813} C_VEL
LIN {X 0,Y 433.665,Z 789.244,A -85,B 0,C 180,E1 -9468.474,E2 -9468.474} C_VEL
LIN {X 0,Y 434.846,Z 764.125,A -85,B 0,C 180,E1 -9472.077,E2 -9472.077} C_VEL
LIN {X 0,Y 436.146,Z 740.784,A -85,B 0,C 180,E1 -9475.41,E2 -9475.41} C_VEL
LIN {X 0,Y 437.202,Z 720.759,A -85,B 0,C 180,E1 -9478.312,E2 -9478.312} C_VEL
LIN {X 0,Y 434.323,Z 707.193,A -85,B 0,C 180,E1 -9480.515,E2 -9480.515} C_VEL
LIN {X 0,Y 432.303,Z 698.63,A -85,B 0,C 180,E1 -9481.995,E2 -9481.995} C_VEL
LIN {X 0,Y 432.288,Z 698.636,A -85,B 0,C 180,E1 -9484.687,E2 -9484.687} C_VEL
LIN {X 0,Y 432.33,Z 698.63,A -85,B 0,C 180,E1 -9488.155,E2 -9488.155} C_VEL
LIN {X 0,Y 432.316,Z 698.632,A -85,B 0,C 180,E1 -9491.804,E2 -9491.804} C_VEL
LIN {X 0,Y 432.328,Z 698.629,A -85,B 0,C 180,E1 -9494.353,E2 -9494.353} C_VEL
LIN {X 0,Y 432.317,Z 698.633,A -85,B 0,C 180,E1 -9497.021,E2 -9497.021} C_VEL
LIN {X 0,Y 432.305,Z 698.634,A -85,B 0,C 180,E1 -9499.83,E2 -9499.83} C_VEL
LIN {X 0,Y 432.314,Z 698.633,A -85,B 0,C 180,E1 -9503.023,E2 -9503.023} C_VEL
LIN {X 0,Y 432.35,Z 698.627,A -85,B 0,C 180,E1 -9506.004,E2 -9506.004} C_VEL
LIN {X 0,Y 432.361,Z 698.63,A -85,B 0,C 180,E1 -9509.492,E2 -9509.492} C_VEL
LIN {X 0,Y 432.352,Z 698.631,A -85,B 0,C 180,E1 -9511.875,E2 -9511.875} C_VEL
LIN {X 0,Y 432.394,Z 698.626,A -85,B 0,C 180,E1 -9515.54,E2 -9515.54} C_VEL
LIN {X 0,Y 432.365,Z 698.63,A -85,B 0,C 180,E1 -9519.047,E2 -9519.047} C_VEL
LIN {X 0,Y 432.408,Z 698.625,A -85,B 0,C 180,E1 -9521.829,E2 -9521.829} C_VEL
LIN {X 0,Y 433.966,Z 702.88,A -85,B 0,C 180,E1 -9522.039,E2 -9522.039} C_VEL
LIN {X 0,Y 437.627,Z 711.777,A -85,B 0,C 180,E1 -9522.451,E2 -9522.451} C_VEL
LIN {X 0,Y 436.647,Z 780.914,A -85,B 0,C 180,E1 -9523.88,E2 -9523.88} C_VEL
LIN {X 0,Y 436.557,Z 792.919,A -85,B 0,C 180,E1 -9524.267,E2 -9524.267} C_VEL
LIN {X 0,Y 436.36,Z 803.943,A -85,B 0,C 180,E1 -9524.768,E2 -9524.768} C_VEL
LIN {X 0,Y 436.054,Z 813.574,A -85,B 0,C 180,E1 -9525.331,E2 -9525.331} C_VEL
LIN {X 0,Y 435.749,Z 822.773,A -85,B 0,C 180,E1 -9526,E2 -9526} C_VEL
LIN {X 0,Y 435.273,Z 832.065,A -85,B 0,C 180,E1 -9526.817,E2 -9526.817} C_VEL
LIN {X 0,Y 434.951,Z 839.819,A -85,B 0,C 180,E1 -9527.638,E2 -9527.638} C_VEL
LIN {X 0,Y 434.542,Z 847.305,A -85,B 0,C 180,E1 -9528.573,E2 -9528.573} C_VEL
LIN {X 0,Y 434.034,Z 855.04,A -85,B 0,C 180,E1 -9529.74,E2 -9529.74} C_VEL
LIN {X 0,Y 433.674,Z 861.42,A -85,B 0,C 180,E1 -9530.909,E2 -9530.909} C_VEL
LIN {X 0,Y 433.371,Z 866.259,A -85,B 0,C 180,E1 -9531.961,E2 -9531.961} C_VEL
LIN {X 0,Y 433.166,Z 870.286,A -85,B 0,C 180,E1 -9533.011,E2 -9533.011} C_VEL
LIN {X 0,Y 432.688,Z 874.571,A -85,B 0,C 180,E1 -9534.407,E2 -9534.407} C_VEL
LIN {X 0,Y 432.495,Z 878.421,A -85,B 0,C 180,E1 -9536.273,E2 -9536.273} C_VEL
LIN {X 0,Y 432.473,Z 879.807,A -85,B 0,C 180,E1 -9537.206,E2 -9537.206} C_VEL
LIN {X 0,Y 432.285,Z 881.147,A -85,B 0,C 180,E1 -9539.068,E2 -9539.068} C_VEL
LIN {X 0,Y 432.25,Z 881.2,A -85,B 0,C 180,E1 -9540,E2 -9540} C_VEL
LIN {X 0,Y 432.252,Z 880.801,A -85,B 0,C 180,E1 -9540.932,E2 -9540.932} C_VEL
LIN {X 0,Y 432.107,Z 878.831,A -85,B 0,C 180,E1 -9542.797,E2 -9542.797} C_VEL
LIN {X 0,Y 432.287,Z 876.181,A -85,B 0,C 180,E1 -9544.196,E2 -9544.196} C_VEL
LIN {X 0,Y 432.476,Z 872.502,A -85,B 0,C 180,E1 -9545.596,E2 -9545.596} C_VEL
LIN {X 0,Y 432.769,Z 867.662,A -85,B 0,C 180,E1 -9546.996,E2 -9546.996} C_VEL
LIN {X 0,Y 433.01,Z 861.536,A -85,B 0,C 180,E1 -9548.4,E2 -9548.4} C_VEL
LIN {X 0,Y 433.338,Z 855.309,A -85,B 0,C 180,E1 -9549.569,E2 -9549.569} C_VEL
LIN {X 0,Y 433.672,Z 847.799,A -85,B 0,C 180,E1 -9550.741,E2 -9550.741} C_VEL
LIN {X 0,Y 434.026,Z 839.688,A -85,B 0,C 180,E1 -9551.796,E2 -9551.796} C_VEL
LIN {X 0,Y 434.409,Z 831.075,A -85,B 0,C 180,E1 -9552.734,E2 -9552.734} C_VEL
LIN {X 0,Y 434.762,Z 822.051,A -85,B 0,C 180,E1 -9553.556,E2 -9553.556} C_VEL
LIN {X 0,Y 435.1,Z 812.747,A -85,B 0,C 180,E1 -9554.258,E2 -9554.258} C_VEL
LIN {X 0,Y 435.322,Z 803.409,A -85,B 0,C 180,E1 -9554.838,E2 -9554.838} C_VEL
LIN {X 0,Y 435.54,Z 792.937,A -85,B 0,C 180,E1 -9555.351,E2 -9555.351} C_VEL
LIN {X 0,Y 435.739,Z 782.516,A -85,B 0,C 180,E1 -9555.734,E2 -9555.734} C_VEL
LIN {X 0,Y 435.813,Z 769.915,A -85,B 0,C 180,E1 -9556.049,E2 -9556.049} C_VEL
LIN {X 0,Y 436.421,Z 710.829,A -85,B 0,C 180,E1 -9557.158,E2 -9557.158} C_VEL
LIN {X 0,Y 432.386,Z 698.624,A -85,B 0,C 180,E1 -9557.556,E2 -9557.556} C_VEL
LIN {X 0,Y 432.354,Z 698.627,A -85,B 0,C 180,E1 -9559.96,E2 -9559.96} C_VEL
LIN {X 0,Y 432.332,Z 698.634,A -85,B 0,C 180,E1 -9562.964,E2 -9562.964} C_VEL
LIN {X 0,Y 432.353,Z 698.631,A -85,B 0,C 180,E1 -9565.001,E2 -9565.001} C_VEL
LIN {X 0,Y 432.36,Z 698.623,A -85,B 0,C 180,E1 -9568.125,E2 -9568.125} C_VEL
LIN {X 0,Y 432.336,Z 698.63,A -85,B 0,C 180,E1 -9571.345,E2 -9571.345} C_VEL
LIN {X 0,Y 432.344,Z 698.63,A -85,B 0,C 180,E1 -9574.677,E2 -9574.677} C_VEL
LIN {X 0,Y 432.346,Z 698.625,A -85,B 0,C 180,E1 -9578.149,E2 -9578.149} C_VEL
LIN {X 0,Y 432.322,Z 698.627,A -85,B 0,C 180,E1 -9581.799,E2 -9581.799} C_VEL
LIN {X 0,Y 432.352,Z 698.623,A -85,B 0,C 180,E1 -9584.345,E2 -9584.345} C_VEL
LIN {X 0,Y 432.318,Z 698.632,A -85,B 0,C 180,E1 -9587.016,E2 -9587.016} C_VEL
LIN {X 0,Y 432.306,Z 698.629,A -85,B 0,C 180,E1 -9589.826,E2 -9589.826} C_VEL
LIN {X 0,Y 432.311,Z 698.633,A -85,B 0,C 180,E1 -9593.018,E2 -9593.018} C_VEL
LIN {X 0,Y 432.347,Z 698.624,A -85,B 0,C 180,E1 -9596,E2 -9596} C_VEL
LIN {X 0,Y 432.347,Z 698.629,A -85,B 0,C 180,E1 -9599.49,E2 -9599.49} C_VEL
LIN {X 0,Y 432.326,Z 698.628,A -85,B 0,C 180,E1 -9601.868,E2 -9601.868} C_VEL
LIN {X 0,Y 432.355,Z 698.63,A -85,B 0,C 180,E1 -9605.546,E2 -9605.546} C_VEL
LIN {X 0,Y 432.335,Z 698.634,A -85,B 0,C 180,E1 -9609.04,E2 -9609.04} C_VEL
LIN {X 0,Y 432.377,Z 698.628,A -85,B 0,C 180,E1 -9611.991,E2 -9611.991} C_VEL
LIN {X 0,Y 437.733,Z 713.574,A -85,B 0,C 180,E1 -9612.49,E2 -9612.49} C_VEL
LIN {X 0,Y 437.076,Z 779.45,A -85,B 0,C 180,E1 -9613.591,E2 -9613.591} C_VEL
LIN {X 0,Y 437.147,Z 787.717,A -85,B 0,C 180,E1 -9613.825,E2 -9613.825} C_VEL
LIN {X 0,Y 435.888,Z 795.36,A -85,B 0,C 180,E1 -9614.052,E2 -9614.052} C_VEL
LIN {X 0,Y 433.344,Z 802.757,A -85,B 0,C 180,E1 -9614.281,E2 -9614.281} C_VEL
LIN {X 0,Y 430.341,Z 811.718,A -85,B 0,C 180,E1 -9614.662,E2 -9614.662} C_VEL
LIN {X 0,Y 429.623,Z 816.957,A -85,B 0,C 180,E1 -9614.986,E2 -9614.986} C_VEL
LIN {X 0,Y 429.09,Z 828.369,A -85,B 0,C 180,E1 -9615.893,E2 -9615.893} C_VEL
LIN {X 0,Y 428.479,Z 838.935,A -85,B 0,C 180,E1 -9616.96,E2 -9616.96} C_VEL
LIN {X 0,Y 427.977,Z 848.404,A -85,B 0,C 180,E1 -9618.149,E2 -9618.149} C_VEL
LIN {X 0,Y 427.343,Z 856.175,A -85,B 0,C 180,E1 -9619.332,E2 -9619.332} C_VEL
LIN {X 0,Y 426.752,Z 863.864,A -85,B 0,C 180,E1 -9620.778,E2 -9620.778} C_VEL
LIN {X 0,Y 426.407,Z 869.511,A -85,B 0,C 180,E1 -9622.102,E2 -9622.102} C_VEL
LIN {X 0,Y 426.037,Z 875.278,A -85,B 0,C 180,E1 -9623.839,E2 -9623.839} C_VEL
LIN {X 0,Y 425.567,Z 878.834,A -85,B 0,C 180,E1 -9625.258,E2 -9625.258} C_VEL
LIN {X 0,Y 425.412,Z 880.659,A -85,B 0,C 180,E1 -9626.205,E2 -9626.205} C_VEL
LIN {X 0,Y 425.397,Z 882.022,A -85,B 0,C 180,E1 -9627.153,E2 -9627.153} C_VEL
LIN {X 0,Y 425.326,Z 883.596,A -85,B 0,C 180,E1 -9629.047,E2 -9629.047} C_VEL
LIN {X 0,Y 425.294,Z 883.832,A -85,B 0,C 180,E1 -9629.994,E2 -9629.994} C_VEL
LIN {X 0,Y 425.43,Z 883.074,A -85,B 0,C 180,E1 -9631.887,E2 -9631.887} C_VEL
LIN {X 0,Y 425.4,Z 880.842,A -85,B 0,C 180,E1 -9633.783,E2 -9633.783} C_VEL
LIN {X 0,Y 425.665,Z 878.035,A -85,B 0,C 180,E1 -9635.203,E2 -9635.203} C_VEL
LIN {X 0,Y 426.062,Z 874.219,A -85,B 0,C 180,E1 -9636.624,E2 -9636.624} C_VEL
LIN {X 0,Y 426.397,Z 868.747,A -85,B 0,C 180,E1 -9638.195,E2 -9638.195} C_VEL
LIN {X 0,Y 426.906,Z 861.942,A -85,B 0,C 180,E1 -9639.708,E2 -9639.708} C_VEL
LIN {X 0,Y 427.546,Z 853.926,A -85,B 0,C 180,E1 -9641.129,E2 -9641.129} C_VEL
LIN {X 0,Y 428.126,Z 845.711,A -85,B 0,C 180,E1 -9642.315,E2 -9642.315} C_VEL
LIN {X 0,Y 428.695,Z 835.558,A -85,B 0,C 180,E1 -9643.503,E2 -9643.503} C_VEL
LIN {X 0,Y 429.358,Z 825.104,A -85,B 0,C 180,E1 -9644.479,E2 -9644.479} C_VEL
LIN {X 0,Y 429.856,Z 813.333,A -85,B 0,C 180,E1 -9645.354,E2 -9645.354} C_VEL
LIN {X 0,Y 430.166,Z 800.832,A -85,B 0,C 180,E1 -9646.051,E2 -9646.051} C_VEL
LIN {X 0,Y 430.343,Z 787.731,A -85,B 0,C 180,E1 -9646.568,E2 -9646.568} C_VEL
LIN {X 0,Y 430.339,Z 775.314,A -85,B 0,C 180,E1 -9646.874,E2 -9646.874} C_VEL
LIN {X 0,Y 430.865,Z 714.201,A -85,B 0,C 180,E1 -9647.902,E2 -9647.902} C_VEL
LIN {X 0,Y 425.37,Z 699.631,A -85,B 0,C 180,E1 -9648.411,E2 -9648.411} C_VEL
LIN {X 0,Y 425.275,Z 699.51,A -85,B 0,C 180,E1 -9651.311,E2 -9651.311} C_VEL
LIN {X 0,Y 425.296,Z 699.505,A -85,B 0,C 180,E1 -9654.649,E2 -9654.649} C_VEL
LIN {X 0,Y 425.319,Z 699.502,A -85,B 0,C 180,E1 -9657.551,E2 -9657.551} C_VEL
LIN {X 0,Y 425.258,Z 699.511,A -85,B 0,C 180,E1 -9660.809,E2 -9660.809} C_VEL
LIN {X 0,Y 425.278,Z 699.505,A -85,B 0,C 180,E1 -9664.281,E2 -9664.281} C_VEL
LIN {X 0,Y 425.249,Z 699.504,A -85,B 0,C 180,E1 -9667.686,E2 -9667.686} C_VEL
LIN {X 0,Y 425.26,Z 699.511,A -85,B 0,C 180,E1 -9670.517,E2 -9670.517} C_VEL
LIN {X 0,Y 425.288,Z 699.509,A -85,B 0,C 180,E1 -9673.355,E2 -9673.355} C_VEL
LIN {X 0,Y 425.284,Z 699.502,A -85,B 0,C 180,E1 -9676.632,E2 -9676.632} C_VEL
LIN {X 0,Y 425.262,Z 699.514,A -85,B 0,C 180,E1 -9679.87,E2 -9679.87} C_VEL
LIN {X 0,Y 425.233,Z 699.514,A -85,B 0,C 180,E1 -9682.481,E2 -9682.481} C_VEL
LIN {X 0,Y 425.249,Z 699.511,A -85,B 0,C 180,E1 -9685.812,E2 -9685.812} C_VEL
LIN {X 0,Y 425.243,Z 699.51,A -85,B 0,C 180,E1 -9689.231,E2 -9689.231} C_VEL
LIN {X 0,Y 425.287,Z 699.51,A -85,B 0,C 180,E1 -9692.438,E2 -9692.438} C_VEL
LIN {X 0,Y 425.287,Z 699.503,A -85,B 0,C 180,E1 -9695.598,E2 -9695.598} C_VEL
LIN {X 0,Y 425.224,Z 699.517,A -85,B 0,C 180,E1 -9698.678,E2 -9698.678} C_VEL
LIN {X 0,Y 425.262,Z 699.505,A -85,B 0,C 180,E1 -9701.699,E2 -9701.699} C_VEL
LIN {X 0,Y 425.289,Z 699.511,A -85,B 0,C 180,E1 -9704.668,E2 -9704.668} C_VEL
LIN {X 0,Y 425.359,Z 699.495,A -85,B 0,C 180,E1 -9707.597,E2 -9707.597} C_VEL
LIN {X 0,Y 425.37,Z 699.497,A -85,B 0,C 180,E1 -9711.448,E2 -9711.448} C_VEL
LIN {X 0,Y 425.503,Z 699.482,A -85,B 0,C 180,E1 -9714.312,E2 -9714.312} C_VEL
LIN {X 0,Y 425.502,Z 699.479,A -85,B 0,C 180,E1 -9718.107,E2 -9718.107} C_VEL
LIN {X 0,Y 425.629,Z 699.465,A -85,B 0,C 180,E1 -9720,E2 -9720} C_VEL
LIN {X 0,Y 425.493,Z 699.48,A -85,B 0,C 180,E1 -9722.84,E2 -9722.84} C_VEL
LIN {X 0,Y 425.504,Z 699.483,A -85,B 0,C 180,E1 -9725.687,E2 -9725.687} C_VEL
LIN {X 0,Y 425.37,Z 699.493,A -85,B 0,C 180,E1 -9728.552,E2 -9728.552} C_VEL
LIN {X 0,Y 425.359,Z 699.497,A -85,B 0,C 180,E1 -9732.403,E2 -9732.403} C_VEL
LIN {X 0,Y 425.327,Z 699.499,A -85,B 0,C 180,E1 -9736.314,E2 -9736.314} C_VEL
LIN {X 0,Y 425.258,Z 699.51,A -85,B 0,C 180,E1 -9739.639,E2 -9739.639} C_VEL
LIN {X 0,Y 425.242,Z 699.514,A -85,B 0,C 180,E1 -9743.369,E2 -9743.369} C_VEL
LIN {X 0,Y 425.284,Z 699.503,A -85,B 0,C 180,E1 -9746.849,E2 -9746.849} C_VEL
LIN {X 0,Y 425.256,Z 699.512,A -85,B 0,C 180,E1 -9749.722,E2 -9749.722} C_VEL
LIN {X 0,Y 425.225,Z 699.513,A -85,B 0,C 180,E1 -9753.053,E2 -9753.053} C_VEL
LIN {X 0,Y 425.228,Z 699.519,A -85,B 0,C 180,E1 -9755.935,E2 -9755.935} C_VEL
LIN {X 0,Y 425.262,Z 699.499,A -85,B 0,C 180,E1 -9759.052,E2 -9759.052} C_VEL
LIN {X 0,Y 425.282,Z 699.51,A -85,B 0,C 180,E1 -9762.652,E2 -9762.652} C_VEL
LIN {X 0,Y 425.289,Z 699.51,A -85,B 0,C 180,E1 -9766.06,E2 -9766.06} C_VEL
LIN {X 0,Y 425.267,Z 699.513,A -85,B 0,C 180,E1 -9768.632,E2 -9768.632} C_VEL
LIN {X 0,Y 425.283,Z 699.508,A -85,B 0,C 180,E1 -9771.111,E2 -9771.111} C_VEL
LIN {X 0,Y 425.264,Z 699.513,A -85,B 0,C 180,E1 -9774.671,E2 -9774.671} C_VEL
LIN {X 0,Y 425.291,Z 699.68,A -85,B 0,C 180,E1 -9777.755,E2 -9777.755} C_VEL
LIN {X 0,Y 429.186,Z 716.281,A -85,B 0,C 180,E1 -9780.586,E2 -9780.586} C_VEL
LIN {X 0,Y 430.276,Z 721.696,A -85,B 0,C 180,E1 -9781.47,E2 -9781.47} C_VEL
LIN {X 0,Y 429.813,Z 732.159,A -85,B 0,C 180,E1 -9783.025,E2 -9783.025} C_VEL
LIN {X 0,Y 428.269,Z 757.861,A -85,B 0,C 180,E1 -9786.777,E2 -9786.777} C_VEL
LIN {X 0,Y 426.968,Z 781.934,A -85,B 0,C 180,E1 -9790.287,E2 -9790.287} C_VEL
LIN {X 0,Y 426.683,Z 788.248,A -85,B 0,C 180,E1 -9791.214,E2 -9791.214} C_VEL
LIN {X 0,Y 430.265,Z 822.606,A -85,B 0,C 180,E1 -9791.973,E2 -9791.973} C_VEL
LIN {X 0,Y 429.404,Z 899.255,A -85,B 0,C 180,E1 -9793.272,E2 -9793.272} C_VEL
LIN {X 0,Y 428.864,Z 912.476,A -85,B 0,C 180,E1 -9793.679,E2 -9793.679} C_VEL
LIN {X 0,Y 428.187,Z 924.662,A -85,B 0,C 180,E1 -9794.233,E2 -9794.233} C_VEL
LIN {X 0,Y 427.432,Z 937.018,A -85,B 0,C 180,E1 -9794.999,E2 -9794.999} C_VEL
LIN {X 0,Y 426.827,Z 947.566,A -85,B 0,C 180,E1 -9795.842,E2 -9795.842} C_VEL
LIN {X 0,Y 426.202,Z 958.249,A -85,B 0,C 180,E1 -9796.902,E2 -9796.902} C_VEL
LIN {X 0,Y 425.512,Z 968.009,A -85,B 0,C 180,E1 -9798.092,E2 -9798.092} C_VEL
LIN {X 0,Y 425.108,Z 976.053,A -85,B 0,C 180,E1 -9799.288,E2 -9799.288} C_VEL
LIN {X 0,Y 424.779,Z 983.938,A -85,B 0,C 180,E1 -9800.724,E2 -9800.724} C_VEL
LIN {X 0,Y 424.618,Z 991.236,A -85,B 0,C 180,E1 -9802.398,E2 -9802.398} C_VEL
LIN {X 0,Y 424.55,Z 995.541,A -85,B 0,C 180,E1 -9803.648,E2 -9803.648} C_VEL
LIN {X 0,Y 424.619,Z 999.848,A -85,B 0,C 180,E1 -9805.26,E2 -9805.26} C_VEL
LIN {X 0,Y 424.66,Z 1001.778,A -85,B 0,C 180,E1 -9806.211,E2 -9806.211} C_VEL
LIN {X 0,Y 424.615,Z 1003.215,A -85,B 0,C 180,E1 -9807.16,E2 -9807.16} C_VEL
LIN {X 0,Y 424.627,Z 1004.245,A -85,B 0,C 180,E1 -9808.109,E2 -9808.109} C_VEL
LIN {X 0,Y 424.635,Z 1004.872,A -85,B 0,C 180,E1 -9809.058,E2 -9809.058} C_VEL
LIN {X 0,Y 424.648,Z 1005.093,A -85,B 0,C 180,E1 -9810.006,E2 -9810.006} C_VEL
LIN {X 0,Y 424.635,Z 1004.864,A -85,B 0,C 180,E1 -9810.955,E2 -9810.955} C_VEL
LIN {X 0,Y 424.628,Z 1004.231,A -85,B 0,C 180,E1 -9811.903,E2 -9811.903} C_VEL
LIN {X 0,Y 424.617,Z 1003.195,A -85,B 0,C 180,E1 -9812.852,E2 -9812.852} C_VEL
LIN {X 0,Y 424.665,Z 1001.751,A -85,B 0,C 180,E1 -9813.802,E2 -9813.802} C_VEL
LIN {X 0,Y 424.58,Z 998.699,A -85,B 0,C 180,E1 -9815.229,E2 -9815.229} C_VEL
LIN {X 0,Y 424.546,Z 994.582,A -85,B 0,C 180,E1 -9816.66,E2 -9816.66} C_VEL
LIN {X 0,Y 424.68,Z 988.273,A -85,B 0,C 180,E1 -9818.332,E2 -9818.332} C_VEL
LIN {X 0,Y 424.876,Z 981.403,A -85,B 0,C 180,E1 -9819.767,E2 -9819.767} C_VEL
LIN {X 0,Y 425.286,Z 972.921,A -85,B 0,C 180,E1 -9821.202,E2 -9821.202} C_VEL
LIN {X 0,Y 425.827,Z 964.254,A -85,B 0,C 180,E1 -9822.395,E2 -9822.395} C_VEL
LIN {X 0,Y 426.46,Z 953.819,A -85,B 0,C 180,E1 -9823.563,E2 -9823.563} C_VEL
LIN {X 0,Y 426.983,Z 943.023,A -85,B 0,C 180,E1 -9824.543,E2 -9824.543} C_VEL
LIN {X 0,Y 427.79,Z 931.529,A -85,B 0,C 180,E1 -9825.367,E2 -9825.367} C_VEL
LIN {X 0,Y 428.467,Z 919.728,A -85,B 0,C 180,E1 -9826.013,E2 -9826.013} C_VEL
LIN {X 0,Y 429.109,Z 906.155,A -85,B 0,C 180,E1 -9826.538,E2 -9826.538} C_VEL
LIN {X 0,Y 429.487,Z 892.636,A -85,B 0,C 180,E1 -9826.86,E2 -9826.86} C_VEL
LIN {X 0,Y 430.198,Z 820.264,A -85,B 0,C 180,E1 -9828.067,E2 -9828.067} C_VEL
LIN {X 0,Y 426.676,Z 788.37,A -85,B 0,C 180,E1 -9828.764,E2 -9828.764} C_VEL
LIN {X 0,Y 427.845,Z 764.845,A -85,B 0,C 180,E1 -9832.203,E2 -9832.203} C_VEL
LIN {X 0,Y 429.177,Z 742.208,A -85,B 0,C 180,E1 -9835.497,E2 -9835.497} C_VEL
LIN {X 0,Y 430.354,Z 723.336,A -85,B 0,C 180,E1 -9838.273,E2 -9838.273} C_VEL
LIN {X 0,Y 429.069,Z 716.136,A -85,B 0,C 180,E1 -9839.437,E2 -9839.437} C_VEL
LIN {X 0,Y 425.26,Z 699.506,A -85,B 0,C 180,E1 -9842.284,E2 -9842.284} C_VEL
LIN {X 0,Y 425.253,Z 699.504,A -85,B 0,C 180,E1 -9845.345,E2 -9845.345} C_VEL
LIN {X 0,Y 425.28,Z 699.51,A -85,B 0,C 180,E1 -9847.699,E2 -9847.699} C_VEL
LIN {X 0,Y 425.261,Z 699.515,A -85,B 0,C 180,E1 -9851.385,E2 -9851.385} C_VEL
LIN {X 0,Y 425.287,Z 699.507,A -85,B 0,C 180,E1 -9854.717,E2 -9854.717} C_VEL
LIN {X 0,Y 425.281,Z 699.508,A -85,B 0,C 180,E1 -9858.048,E2 -9858.048} C_VEL
LIN {X 0,Y 425.293,Z 699.508,A -85,B 0,C 180,E1 -9861.101,E2 -9861.101} C_VEL
LIN {X 0,Y 425.31,Z 699.504,A -85,B 0,C 180,E1 -9864.665,E2 -9864.665} C_VEL
LIN {X 0,Y 425.28,Z 699.507,A -85,B 0,C 180,E1 -9868.074,E2 -9868.074} C_VEL
LIN {X 0,Y 425.322,Z 699.507,A -85,B 0,C 180,E1 -9871.367,E2 -9871.367} C_VEL
LIN {X 0,Y 425.285,Z 699.509,A -85,B 0,C 180,E1 -9874.554,E2 -9874.554} C_VEL
LIN {X 0,Y 425.299,Z 699.507,A -85,B 0,C 180,E1 -9876.634,E2 -9876.634} C_VEL
LIN {X 0,Y 425.311,Z 699.509,A -85,B 0,C 180,E1 -9879.695,E2 -9879.695} C_VEL
LIN {X 0,Y 425.371,Z 699.509,A -85,B 0,C 180,E1 -9881.439,E2 -9881.439} C_VEL
LIN {X 0,Y 426.467,Z 702.535,A -85,B 0,C 180,E1 -9881.582,E2 -9881.582} C_VEL
LIN {X 0,Y 431.069,Z 713.524,A -85,B 0,C 180,E1 -9882.116,E2 -9882.116} C_VEL
LIN {X 0,Y 429.918,Z 783.281,A -85,B 0,C 180,E1 -9883.621,E2 -9883.621} C_VEL
LIN {X 0,Y 429.868,Z 794.916,A -85,B 0,C 180,E1 -9884.015,E2 -9884.015} C_VEL
LIN {X 0,Y 429.652,Z 805.751,A -85,B 0,C 180,E1 -9884.524,E2 -9884.524} C_VEL
LIN {X 0,Y 429.34,Z 815.048,A -85,B 0,C 180,E1 -9885.081,E2 -9885.081} C_VEL
LIN {X 0,Y 429.02,Z 824.377,A -85,B 0,C 180,E1 -9885.775,E2 -9885.775} C_VEL
LIN {X 0,Y 428.508,Z 833.566,A -85,B 0,C 180,E1 -9886.605,E2 -9886.605} C_VEL
LIN {X 0,Y 428.167,Z 841.24,A -85,B 0,C 180,E1 -9887.438,E2 -9887.438} C_VEL
LIN {X 0,Y 427.722,Z 848.661,A -85,B 0,C 180,E1 -9888.388,E2 -9888.388} C_VEL
LIN {X 0,Y 427.19,Z 856.35,A -85,B 0,C 180,E1 -9889.574,E2 -9889.574} C_VEL
LIN {X 0,Y 426.789,Z 862.712,A -85,B 0,C 180,E1 -9890.761,E2 -9890.761} C_VEL
LIN {X 0,Y 426.472,Z 867.332,A -85,B 0,C 180,E1 -9891.778,E2 -9891.778} C_VEL
LIN {X 0,Y 426.238,Z 871.548,A -85,B 0,C 180,E1 -9892.896,E2 -9892.896} C_VEL
LIN {X 0,Y 425.73,Z 875.8,A -85,B 0,C 180,E1 -9894.316,E2 -9894.316} C_VEL
LIN {X 0,Y 425.634,Z 877.913,A -85,B 0,C 180,E1 -9895.264,E2 -9895.264} C_VEL
LIN {X 0,Y 425.478,Z 880.956,A -85,B 0,C 180,E1 -9897.16,E2 -9897.16} C_VEL
LIN {X 0,Y 425.272,Z 882.249,A -85,B 0,C 180,E1 -9899.053,E2 -9899.053} C_VEL
LIN {X 0,Y 425.233,Z 882.262,A -85,B 0,C 180,E1 -9900,E2 -9900} C_VEL
LIN {X 0,Y 425.236,Z 881.831,A -85,B 0,C 180,E1 -9900.947,E2 -9900.947} C_VEL
LIN {X 0,Y 425.082,Z 879.799,A -85,B 0,C 180,E1 -9902.843,E2 -9902.843} C_VEL
LIN {X 0,Y 425.271,Z 877.093,A -85,B 0,C 180,E1 -9904.265,E2 -9904.265} C_VEL
LIN {X 0,Y 425.48,Z 873.343,A -85,B 0,C 180,E1 -9905.688,E2 -9905.688} C_VEL
LIN {X 0,Y 425.78,Z 868.429,A -85,B 0,C 180,E1 -9907.111,E2 -9907.111} C_VEL
LIN {X 0,Y 426.011,Z 862.221,A -85,B 0,C 180,E1 -9908.539,E2 -9908.539} C_VEL
LIN {X 0,Y 426.374,Z 855.906,A -85,B 0,C 180,E1 -9909.727,E2 -9909.727} C_VEL
LIN {X 0,Y 426.717,Z 848.293,A -85,B 0,C 180,E1 -9910.918,E2 -9910.918} C_VEL
LIN {X 0,Y 427.086,Z 840.067,A -85,B 0,C 180,E1 -9911.991,E2 -9911.991} C_VEL
LIN {X 0,Y 427.448,Z 832.532,A -85,B 0,C 180,E1 -9912.825,E2 -9912.825} C_VEL
LIN {X 0,Y 427.789,Z 823.658,A -85,B 0,C 180,E1 -9913.655,E2 -9913.655} C_VEL
LIN {X 0,Y 428.163,Z 813.672,A -85,B 0,C 180,E1 -9914.423,E2 -9914.423} C_VEL
LIN {X 0,Y 428.399,Z 804.237,A -85,B 0,C 180,E1 -9915.017,E2 -9915.017} C_VEL
LIN {X 0,Y 428.626,Z 793.58,A -85,B 0,C 180,E1 -9915.544,E2 -9915.544} C_VEL
LIN {X 0,Y 428.841,Z 783.046,A -85,B 0,C 180,E1 -9915.933,E2 -9915.933} C_VEL
LIN {X 0,Y 428.909,Z 770.44,A -85,B 0,C 180,E1 -9916.25,E2 -9916.25} C_VEL
LIN {X 0,Y 429.534,Z 712.234,A -85,B 0,C 180,E1 -9917.372,E2 -9917.372} C_VEL
LIN {X 0,Y 425.332,Z 699.503,A -85,B 0,C 180,E1 -9917.79,E2 -9917.79} C_VEL
LIN {X 0,Y 425.311,Z 699.506,A -85,B 0,C 180,E1 -9920.305,E2 -9920.305} C_VEL
LIN {X 0,Y 425.299,Z 699.506,A -85,B 0,C 180,E1 -9923.366,E2 -9923.366} C_VEL
LIN {X 0,Y 425.316,Z 699.505,A -85,B 0,C 180,E1 -9926.497,E2 -9926.497} C_VEL
LIN {X 0,Y 425.303,Z 699.504,A -85,B 0,C 180,E1 -9929.719,E2 -9929.719} C_VEL
LIN {X 0,Y 425.287,Z 699.509,A -85,B 0,C 180,E1 -9933.048,E2 -9933.048} C_VEL
LIN {X 0,Y 425.297,Z 699.503,A -85,B 0,C 180,E1 -9935.926,E2 -9935.926} C_VEL
LIN {X 0,Y 425.279,Z 699.51,A -85,B 0,C 180,E1 -9939.035,E2 -9939.035} C_VEL
LIN {X 0,Y 425.275,Z 699.508,A -85,B 0,C 180,E1 -9942.653,E2 -9942.653} C_VEL
LIN {X 0,Y 425.303,Z 699.505,A -85,B 0,C 180,E1 -9945.281,E2 -9945.281} C_VEL
LIN {X 0,Y 425.265,Z 699.508,A -85,B 0,C 180,E1 -9948.615,E2 -9948.615} C_VEL
LIN {X 0,Y 425.293,Z 699.507,A -85,B 0,C 180,E1 -9951.096,E2 -9951.096} C_VEL
LIN {X 0,Y 425.307,Z 699.502,A -85,B 0,C 180,E1 -9954.66,E2 -9954.66} C_VEL
LIN {X 0,Y 425.262,Z 699.507,A -85,B 0,C 180,E1 -9958.068,E2 -9958.068} C_VEL
LIN {X 0,Y 425.307,Z 699.507,A -85,B 0,C 180,E1 -9961.361,E2 -9961.361} C_VEL
LIN {X 0,Y 425.257,Z 699.51,A -85,B 0,C 180,E1 -9964.547,E2 -9964.547} C_VEL
LIN {X 0,Y 425.304,Z 699.508,A -85,B 0,C 180,E1 -9967.727,E2 -9967.727} C_VEL
LIN {X 0,Y 425.339,Z 699.506,A -85,B 0,C 180,E1 -9971.448,E2 -9971.448} C_VEL
LIN {X 0,Y 425.324,Z 699.508,A -85,B 0,C 180,E1 -9971.666,E2 -9971.666} C_VEL
LIN {X 0,Y 428.289,Z 707.593,A -85,B 0,C 180,E1 -9971.962,E2 -9971.962} C_VEL
LIN {X 0,Y 430.853,Z 714.296,A -85,B 0,C 180,E1 -9972.195,E2 -9972.195} C_VEL
LIN {X 0,Y 430.335,Z 780.476,A -85,B 0,C 180,E1 -9973.327,E2 -9973.327} C_VEL
LIN {X 0,Y 430.349,Z 793.283,A -85,B 0,C 180,E1 -9973.724,E2 -9973.724} C_VEL
LIN {X 0,Y 430.053,Z 805.681,A -85,B 0,C 180,E1 -9974.291,E2 -9974.291} C_VEL
LIN {X 0,Y 429.623,Z 816.957,A -85,B 0,C 180,E1 -9974.986,E2 -9974.986} C_VEL
LIN {X 0,Y 428.908,Z 820.494,A -85,B 0,C 180,E1 -9975.213,E2 -9975.213} C_VEL
LIN {X 0,Y 425.919,Z 826.094,A -85,B 0,C 180,E1 -9975.528,E2 -9975.528} C_VEL
LIN {X 0,Y 422.837,Z 831.503,A -85,B 0,C 180,E1 -9975.888,E2 -9975.888} C_VEL
LIN {X 0,Y 421.986,Z 834.739,A -85,B 0,C 180,E1 -9976.183,E2 -9976.183} C_VEL
LIN {X 0,Y 421.37,Z 843.976,A -85,B 0,C 180,E1 -9977.227,E2 -9977.227} C_VEL
LIN {X 0,Y 420.854,Z 852.681,A -85,B 0,C 180,E1 -9978.434,E2 -9978.434} C_VEL
LIN {X 0,Y 420.112,Z 861.193,A -85,B 0,C 180,E1 -9979.878,E2 -9979.878} C_VEL
LIN {X 0,Y 419.503,Z 867.963,A -85,B 0,C 180,E1 -9981.322,E2 -9981.322} C_VEL
LIN {X 0,Y 419.281,Z 873.336,A -85,B 0,C 180,E1 -9982.772,E2 -9982.772} C_VEL
LIN {X 0,Y 418.752,Z 877.6,A -85,B 0,C 180,E1 -9984.215,E2 -9984.215} C_VEL
LIN {X 0,Y 418.563,Z 879.837,A -85,B 0,C 180,E1 -9985.178,E2 -9985.178} C_VEL
LIN {X 0,Y 418.399,Z 881.662,A -85,B 0,C 180,E1 -9986.141,E2 -9986.141} C_VEL
LIN {X 0,Y 418.379,Z 883.025,A -85,B 0,C 180,E1 -9987.105,E2 -9987.105} C_VEL
LIN {X 0,Y 418.373,Z 883.992,A -85,B 0,C 180,E1 -9988.068,E2 -9988.068} C_VEL
LIN {X 0,Y 418.27,Z 884.834,A -85,B 0,C 180,E1 -9989.994,E2 -9989.994} C_VEL
LIN {X 0,Y 418.41,Z 884.076,A -85,B 0,C 180,E1 -9991.919,E2 -9991.919} C_VEL
LIN {X 0,Y 418.387,Z 881.844,A -85,B 0,C 180,E1 -9993.846,E2 -9993.846} C_VEL
LIN {X 0,Y 418.667,Z 879.037,A -85,B 0,C 180,E1 -9995.291,E2 -9995.291} C_VEL
LIN {X 0,Y 419.087,Z 875.22,A -85,B 0,C 180,E1 -9996.735,E2 -9996.735} C_VEL
LIN {X 0,Y 419.442,Z 869.748,A -85,B 0,C 180,E1 -9998.332,E2 -9998.332} C_VEL
LIN {X 0,Y 419.981,Z 862.942,A -85,B 0,C 180,E1 -9999.869,E2 -9999.869} C_VEL
LIN {X 0,Y 420.655,Z 854.925,A -85,B 0,C 180,E1 -10001.314,E2 -10001.314} C_VEL
LIN {X 0,Y 421.263,Z 846.711,A -85,B 0,C 180,E1 -10002.519,E2 -10002.519} C_VEL
LIN {X 0,Y 421.864,Z 836.556,A -85,B 0,C 180,E1 -10003.725,E2 -10003.725} C_VEL
LIN {X 0,Y 422.557,Z 826.102,A -85,B 0,C 180,E1 -10004.717,E2 -10004.717} C_VEL
LIN {X 0,Y 423.085,Z 814.328,A -85,B 0,C 180,E1 -10005.606,E2 -10005.606} C_VEL
LIN {X 0,Y 423.412,Z 801.826,A -85,B 0,C 180,E1 -10006.314,E2 -10006.314} C_VEL
LIN {X 0,Y 423.592,Z 788.723,A -85,B 0,C 180,E1 -10006.84,E2 -10006.84} C_VEL
LIN {X 0,Y 423.6,Z 776.293,A -85,B 0,C 180,E1 -10007.15,E2 -10007.15} C_VEL
LIN {X 0,Y 424.13,Z 715.771,A -85,B 0,C 180,E1 -10008.186,E2 -10008.186} C_VEL
LIN {X 0,Y 418.327,Z 700.503,A -85,B 0,C 180,E1 -10008.735,E2 -10008.735} C_VEL
LIN {X 0,Y 418.218,Z 700.384,A -85,B 0,C 180,E1 -10012.443,E2 -10012.443} C_VEL
LIN {X 0,Y 418.262,Z 700.382,A -85,B 0,C 180,E1 -10014.857,E2 -10014.857} C_VEL
LIN {X 0,Y 418.263,Z 700.378,A -85,B 0,C 180,E1 -10018.056,E2 -10018.056} C_VEL
LIN {X 0,Y 418.181,Z 700.396,A -85,B 0,C 180,E1 -10021.389,E2 -10021.389} C_VEL
LIN {X 0,Y 418.232,Z 700.383,A -85,B 0,C 180,E1 -10024.573,E2 -10024.573} C_VEL
LIN {X 0,Y 418.199,Z 700.38,A -85,B 0,C 180,E1 -10027.828,E2 -10027.828} C_VEL
LIN {X 0,Y 418.226,Z 700.388,A -85,B 0,C 180,E1 -10030.936,E2 -10030.936} C_VEL
LIN {X 0,Y 418.239,Z 700.38,A -85,B 0,C 180,E1 -10033.733,E2 -10033.733} C_VEL
LIN {X 0,Y 418.235,Z 700.38,A -85,B 0,C 180,E1 -10036.452,E2 -10036.452} C_VEL
LIN {X 0,Y 418.217,Z 700.389,A -85,B 0,C 180,E1 -10039.117,E2 -10039.117} C_VEL
LIN {X 0,Y 418.185,Z 700.395,A -85,B 0,C 180,E1 -10042.159,E2 -10042.159} C_VEL
LIN {X 0,Y 418.208,Z 700.387,A -85,B 0,C 180,E1 -10045.414,E2 -10045.414} C_VEL
LIN {X 0,Y 418.162,Z 700.394,A -85,B 0,C 180,E1 -10048.6,E2 -10048.6} C_VEL
LIN {X 0,Y 418.232,Z 700.383,A -85,B 0,C 180,E1 -10051.932,E2 -10051.932} C_VEL
LIN {X 0,Y 418.225,Z 700.382,A -85,B 0,C 180,E1 -10055.158,E2 -10055.158} C_VEL
LIN {X 0,Y 418.166,Z 700.396,A -85,B 0,C 180,E1 -10058.3,E2 -10058.3} C_VEL
LIN {X 0,Y 418.213,Z 700.383,A -85,B 0,C 180,E1 -10061.38,E2 -10061.38} C_VEL
LIN {X 0,Y 418.242,Z 700.384,A -85,B 0,C 180,E1 -10064.404,E2 -10064.404} C_VEL
LIN {X 0,Y 418.299,Z 700.375,A -85,B 0,C 180,E1 -10067.384,E2 -10067.384} C_VEL
LIN {X 0,Y 418.29,Z 700.374,A -85,B 0,C 180,E1 -10070.327,E2 -10070.327} C_VEL
LIN {X 0,Y 418.421,Z 700.365,A -85,B 0,C 180,E1 -10073.248,E2 -10073.248} C_VEL
LIN {X 0,Y 418.277,Z 700.376,A -85,B 0,C 180,E1 -10075.181,E2 -10075.181} C_VEL
LIN {X 0,Y 418.472,Z 700.355,A -85,B 0,C 180,E1 -10078.075,E2 -10078.075} C_VEL
LIN {X 0,Y 418.599,Z 700.341,A -85,B 0,C 180,E1 -10080,E2 -10080} C_VEL
LIN {X 0,Y 418.447,Z 700.357,A -85,B 0,C 180,E1 -10082.888,E2 -10082.888} C_VEL
LIN {X 0,Y 418.459,Z 700.36,A -85,B 0,C 180,E1 -10085.783,E2 -10085.783} C_VEL
LIN {X 0,Y 418.328,Z 700.371,A -85,B 0,C 180,E1 -10088.697,E2 -10088.697} C_VEL
LIN {X 0,Y 418.265,Z 700.385,A -85,B 0,C 180,E1 -10091.632,E2 -10091.632} C_VEL
LIN {X 0,Y 418.242,Z 700.383,A -85,B 0,C 180,E1 -10094.599,E2 -10094.599} C_VEL
LIN {X 0,Y 418.218,Z 700.393,A -85,B 0,C 180,E1 -10097.607,E2 -10097.607} C_VEL
LIN {X 0,Y 418.181,Z 700.384,A -85,B 0,C 180,E1 -10100.667,E2 -10100.667} C_VEL
LIN {X 0,Y 418.224,Z 700.39,A -85,B 0,C 180,E1 -10103.785,E2 -10103.785} C_VEL
LIN {X 0,Y 418.246,Z 700.38,A -85,B 0,C 180,E1 -10107.075,E2 -10107.075} C_VEL
LIN {X 0,Y 418.201,Z 700.387,A -85,B 0,C 180,E1 -10110.276,E2 -10110.276} C_VEL
LIN {X 0,Y 418.191,Z 700.393,A -85,B 0,C 180,E1 -10113.683,E2 -10113.683} C_VEL
LIN {X 0,Y 418.192,Z 700.388,A -85,B 0,C 180,E1 -10117.229,E2 -10117.229} C_VEL
LIN {X 0,Y 418.215,Z 700.379,A -85,B 0,C 180,E1 -10119.686,E2 -10119.686} C_VEL
LIN {X 0,Y 418.235,Z 700.389,A -85,B 0,C 180,E1 -10122.336,E2 -10122.336} C_VEL
LIN {X 0,Y 418.228,Z 700.386,A -85,B 0,C 180,E1 -10125.121,E2 -10125.121} C_VEL
LIN {X 0,Y 418.249,Z 700.379,A -85,B 0,C 180,E1 -10127.78,E2 -10127.78} C_VEL
LIN {X 0,Y 418.226,Z 700.387,A -85,B 0,C 180,E1 -10131.567,E2 -10131.567} C_VEL
LIN {X 0,Y 418.225,Z 700.385,A -85,B 0,C 180,E1 -10135.166,E2 -10135.166} C_VEL
LIN {X 0,Y 418.227,Z 700.462,A -85,B 0,C 180,E1 -10137.424,E2 -10137.424} C_VEL
LIN {X 0,Y 422.046,Z 716.689,A -85,B 0,C 180,E1 -10140.254,E2 -10140.254} C_VEL
LIN {X 0,Y 423.457,Z 724.147,A -85,B 0,C 180,E1 -10141.491,E2 -10141.491} C_VEL
LIN {X 0,Y 422.344,Z 741.511,A -85,B 0,C 180,E1 -10144.092,E2 -10144.092} C_VEL
LIN {X 0,Y 421.011,Z 763.987,A -85,B 0,C 180,E1 -10147.43,E2 -10147.43} C_VEL
LIN {X 0,Y 419.739,Z 787.204,A -85,B 0,C 180,E1 -10150.888,E2 -10150.888} C_VEL
LIN {X 0,Y 423.486,Z 822.768,A -85,B 0,C 180,E1 -10151.695,E2 -10151.695} C_VEL
LIN {X 0,Y 422.622,Z 898.255,A -85,B 0,C 180,E1 -10152.996,E2 -10152.996} C_VEL
LIN {X 0,Y 422.048,Z 911.47,A -85,B 0,C 180,E1 -10153.408,E2 -10153.408} C_VEL
LIN {X 0,Y 421.346,Z 923.653,A -85,B 0,C 180,E1 -10153.971,E2 -10153.971} C_VEL
LIN {X 0,Y 420.557,Z 936.006,A -85,B 0,C 180,E1 -10154.748,E2 -10154.748} C_VEL
LIN {X 0,Y 419.86,Z 946.411,A -85,B 0,C 180,E1 -10155.59,E2 -10155.59} C_VEL
LIN {X 0,Y 419.167,Z 957.221,A -85,B 0,C 180,E1 -10156.679,E2 -10156.679} C_VEL
LIN {X 0,Y 418.669,Z 965.178,A -85,B 0,C 180,E1 -10157.649,E2 -10157.649} C_VEL
LIN {X 0,Y 418.081,Z 975.034,A -85,B 0,C 180,E1 -10159.106,E2 -10159.106} C_VEL
LIN {X 0,Y 417.729,Z 982.92,A -85,B 0,C 180,E1 -10160.566,E2 -10160.566} C_VEL
LIN {X 0,Y 417.547,Z 990.219,A -85,B 0,C 180,E1 -10162.268,E2 -10162.268} C_VEL
LIN {X 0,Y 417.486,Z 994.829,A -85,B 0,C 180,E1 -10163.639,E2 -10163.639} C_VEL
LIN {X 0,Y 417.575,Z 998.84,A -85,B 0,C 180,E1 -10165.179,E2 -10165.179} C_VEL
LIN {X 0,Y 417.624,Z 1000.773,A -85,B 0,C 180,E1 -10166.147,E2 -10166.147} C_VEL
LIN {X 0,Y 417.574,Z 1002.209,A -85,B 0,C 180,E1 -10167.112,E2 -10167.112} C_VEL
LIN {X 0,Y 417.589,Z 1003.24,A -85,B 0,C 180,E1 -10168.078,E2 -10168.078} C_VEL
LIN {X 0,Y 417.603,Z 1003.869,A -85,B 0,C 180,E1 -10169.042,E2 -10169.042} C_VEL
LIN {X 0,Y 417.62,Z 1004.091,A -85,B 0,C 180,E1 -10170.006,E2 -10170.006} C_VEL
LIN {X 0,Y 417.603,Z 1003.861,A -85,B 0,C 180,E1 -10170.971,E2 -10170.971} C_VEL
LIN {X 0,Y 417.59,Z 1003.226,A -85,B 0,C 180,E1 -10171.935,E2 -10171.935} C_VEL
LIN {X 0,Y 417.576,Z 1002.189,A -85,B 0,C 180,E1 -10172.9,E2 -10172.9} C_VEL
LIN {X 0,Y 417.629,Z 1000.745,A -85,B 0,C 180,E1 -10173.866,E2 -10173.866} C_VEL
LIN {X 0,Y 417.506,Z 997.685,A -85,B 0,C 180,E1 -10175.318,E2 -10175.318} C_VEL
LIN {X 0,Y 417.482,Z 993.566,A -85,B 0,C 180,E1 -10176.773,E2 -10176.773} C_VEL
LIN {X 0,Y 417.62,Z 987.254,A -85,B 0,C 180,E1 -10178.474,E2 -10178.474} C_VEL
LIN {X 0,Y 417.823,Z 980.381,A -85,B 0,C 180,E1 -10179.934,E2 -10179.934} C_VEL
LIN {X 0,Y 418.265,Z 971.898,A -85,B 0,C 180,E1 -10181.393,E2 -10181.393} C_VEL
LIN {X 0,Y 418.86,Z 963.234,A -85,B 0,C 180,E1 -10182.605,E2 -10182.605} C_VEL
LIN {X 0,Y 419.439,Z 953.746,A -85,B 0,C 180,E1 -10183.696,E2 -10183.696} C_VEL
LIN {X 0,Y 420.076,Z 942.001,A -85,B 0,C 180,E1 -10184.787,E2 -10184.787} C_VEL
LIN {X 0,Y 420.896,Z 930.504,A -85,B 0,C 180,E1 -10185.625,E2 -10185.625} C_VEL
LIN {X 0,Y 421.595,Z 918.701,A -85,B 0,C 180,E1 -10186.281,E2 -10186.281} C_VEL
LIN {X 0,Y 422.3,Z 905.132,A -85,B 0,C 180,E1 -10186.813,E2 -10186.813} C_VEL
LIN {X 0,Y 422.708,Z 891.606,A -85,B 0,C 180,E1 -10187.139,E2 -10187.139} C_VEL
LIN {X 0,Y 423.385,Z 820.721,A -85,B 0,C 180,E1 -10188.342,E2 -10188.342} C_VEL
LIN {X 0,Y 419.724,Z 787.138,A -85,B 0,C 180,E1 -10189.117,E2 -10189.117} C_VEL
LIN {X 0,Y 421.091,Z 762.346,A -85,B 0,C 180,E1 -10192.81,E2 -10192.81} C_VEL
LIN {X 0,Y 422.386,Z 740.59,A -85,B 0,C 180,E1 -10196.039,E2 -10196.039} C_VEL
LIN {X 0,Y 423.417,Z 724.074,A -85,B 0,C 180,E1 -10198.517,E2 -10198.517} C_VEL
LIN {X 0,Y 420.838,Z 711.506,A -85,B 0,C 180,E1 -10200.626,E2 -10200.626} C_VEL
LIN {X 0,Y 418.219,Z 700.382,A -85,B 0,C 180,E1 -10202.588,E2 -10202.588} C_VEL
LIN {X 0,Y 418.218,Z 700.379,A -85,B 0,C 180,E1 -10206.232,E2 -10206.232} C_VEL
LIN {X 0,Y 418.212,Z 700.394,A -85,B 0,C 180,E1 -10209.374,E2 -10209.374} C_VEL
LIN {X 0,Y 418.199,Z 700.389,A -85,B 0,C 180,E1 -10212.316,E2 -10212.316} C_VEL
LIN {X 0,Y 418.244,Z 700.387,A -85,B 0,C 180,E1 -10215.11,E2 -10215.11} C_VEL
LIN {X 0,Y 418.235,Z 700.387,A -85,B 0,C 180,E1 -10217.766,E2 -10217.766} C_VEL
LIN {X 0,Y 418.251,Z 700.387,A -85,B 0,C 180,E1 -10221.558,E2 -10221.558} C_VEL
LIN {X 0,Y 418.267,Z 700.384,A -85,B 0,C 180,E1 -10225.16,E2 -10225.16} C_VEL
LIN {X 0,Y 418.261,Z 700.386,A -85,B 0,C 180,E1 -10227.473,E2 -10227.473} C_VEL
LIN {X 0,Y 418.28,Z 700.384,A -85,B 0,C 180,E1 -10230.899,E2 -10230.899} C_VEL
LIN {X 0,Y 418.248,Z 700.386,A -85,B 0,C 180,E1 -10234.094,E2 -10234.094} C_VEL
LIN {X 0,Y 418.248,Z 700.388,A -85,B 0,C 180,E1 -10237.264,E2 -10237.264} C_VEL
LIN {X 0,Y 418.338,Z 700.442,A -85,B 0,C 180,E1 -10240.991,E2 -10240.991} C_VEL
LIN {X 0,Y 419.411,Z 703.328,A -85,B 0,C 180,E1 -10241.139,E2 -10241.139} C_VEL
LIN {X 0,Y 424.605,Z 715.451,A -85,B 0,C 180,E1 -10241.78,E2 -10241.78} C_VEL
LIN {X 0,Y 423.28,Z 784.03,A -85,B 0,C 180,E1 -10243.295,E2 -10243.295} C_VEL
LIN {X 0,Y 423.235,Z 795.682,A -85,B 0,C 180,E1 -10243.696,E2 -10243.696} C_VEL
LIN {X 0,Y 423.004,Z 806.544,A -85,B 0,C 180,E1 -10244.213,E2 -10244.213} C_VEL
LIN {X 0,Y 422.656,Z 816.439,A -85,B 0,C 180,E1 -10244.818,E2 -10244.818} C_VEL
LIN {X 0,Y 422.294,Z 825.985,A -85,B 0,C 180,E1 -10245.544,E2 -10245.544} C_VEL
LIN {X 0,Y 421.765,Z 835.114,A -85,B 0,C 180,E1 -10246.387,E2 -10246.387} C_VEL
LIN {X 0,Y 421.409,Z 842.739,A -85,B 0,C 180,E1 -10247.234,E2 -10247.234} C_VEL
LIN {X 0,Y 420.923,Z 850.123,A -85,B 0,C 180,E1 -10248.198,E2 -10248.198} C_VEL
LIN {X 0,Y 420.358,Z 857.763,A -85,B 0,C 180,E1 -10249.402,E2 -10249.402} C_VEL
LIN {X 0,Y 420.054,Z 862.947,A -85,B 0,C 180,E1 -10250.368,E2 -10250.368} C_VEL
LIN {X 0,Y 419.603,Z 868.414,A -85,B 0,C 180,E1 -10251.584,E2 -10251.584} C_VEL
LIN {X 0,Y 419.308,Z 872.81,A -85,B 0,C 180,E1 -10252.778,E2 -10252.778} C_VEL
LIN {X 0,Y 418.772,Z 877.025,A -85,B 0,C 180,E1 -10254.221,E2 -10254.221} C_VEL
LIN {X 0,Y 418.682,Z 879.129,A -85,B 0,C 180,E1 -10255.186,E2 -10255.186} C_VEL
LIN {X 0,Y 418.484,Z 882.108,A -85,B 0,C 180,E1 -10257.112,E2 -10257.112} C_VEL
LIN {X 0,Y 418.261,Z 883.36,A -85,B 0,C 180,E1 -10259.037,E2 -10259.037} C_VEL
LIN {X 0,Y 418.216,Z 883.331,A -85,B 0,C 180,E1 -10260,E2 -10260} C_VEL
LIN {X 0,Y 418.219,Z 882.872,A -85,B 0,C 180,E1 -10260.963,E2 -10260.963} C_VEL
LIN {X 0,Y 418.055,Z 880.748,A -85,B 0,C 180,E1 -10262.891,E2 -10262.891} C_VEL
LIN {X 0,Y 418.255,Z 877.972,A -85,B 0,C 180,E1 -10264.337,E2 -10264.337} C_VEL
LIN {X 0,Y 418.485,Z 874.144,A -85,B 0,C 180,E1 -10265.783,E2 -10265.783} C_VEL
LIN {X 0,Y 418.792,Z 869.15,A -85,B 0,C 180,E1 -10267.231,E2 -10267.231} C_VEL
LIN {X 0,Y 419.014,Z 864.005,A -85,B 0,C 180,E1 -10268.448,E2 -10268.448} C_VEL
LIN {X 0,Y 419.292,Z 857.887,A -85,B 0,C 180,E1 -10269.649,E2 -10269.649} C_VEL
LIN {X 0,Y 419.701,Z 850.438,A -85,B 0,C 180,E1 -10270.859,E2 -10270.859} C_VEL
LIN {X 0,Y 420.036,Z 842.414,A -85,B 0,C 180,E1 -10271.95,E2 -10271.95} C_VEL
LIN {X 0,Y 420.459,Z 833.914,A -85,B 0,C 180,E1 -10272.919,E2 -10272.919} C_VEL
LIN {X 0,Y 420.87,Z 823.98,A -85,B 0,C 180,E1 -10273.856,E2 -10273.856} C_VEL
LIN {X 0,Y 421.191,Z 814.815,A -85,B 0,C 180,E1 -10274.572,E2 -10274.572} C_VEL
LIN {X 0,Y 421.483,Z 804.949,A -85,B 0,C 180,E1 -10275.201,E2 -10275.201} C_VEL
LIN {X 0,Y 421.72,Z 794.096,A -85,B 0,C 180,E1 -10275.743,E2 -10275.743} C_VEL
LIN {X 0,Y 421.942,Z 783.447,A -85,B 0,C 180,E1 -10276.138,E2 -10276.138} C_VEL
LIN {X 0,Y 422.002,Z 770.318,A -85,B 0,C 180,E1 -10276.47,E2 -10276.47} C_VEL
LIN {X 0,Y 422.663,Z 713.561,A -85,B 0,C 180,E1 -10277.595,E2 -10277.595} C_VEL
LIN {X 0,Y 418.33,Z 700.376,A -85,B 0,C 180,E1 -10278.027,E2 -10278.027} C_VEL
LIN {X 0,Y 418.266,Z 700.387,A -85,B 0,C 180,E1 -10280.662,E2 -10280.662} C_VEL
LIN {X 0,Y 418.29,Z 700.377,A -85,B 0,C 180,E1 -10283.781,E2 -10283.781} C_VEL
LIN {X 0,Y 418.242,Z 700.386,A -85,B 0,C 180,E1 -10287.046,E2 -10287.046} C_VEL
LIN {X 0,Y 418.26,Z 700.382,A -85,B 0,C 180,E1 -10290.271,E2 -10290.271} C_VEL
LIN {X 0,Y 418.25,Z 700.381,A -85,B 0,C 180,E1 -10293.677,E2 -10293.677} C_VEL
LIN {X 0,Y 418.255,Z 700.385,A -85,B 0,C 180,E1 -10297.223,E2 -10297.223} C_VEL
LIN {X 0,Y 418.225,Z 700.39,A -85,B 0,C 180,E1 -10300.865,E2 -10300.865} C_VEL
LIN {X 0,Y 418.221,Z 700.383,A -85,B 0,C 180,E1 -10303.726,E2 -10303.726} C_VEL
LIN {X 0,Y 418.216,Z 700.384,A -85,B 0,C 180,E1 -10306.445,E2 -10306.445} C_VEL
LIN {X 0,Y 418.225,Z 700.387,A -85,B 0,C 180,E1 -10309.13,E2 -10309.13} C_VEL
LIN {X 0,Y 418.249,Z 700.382,A -85,B 0,C 180,E1 -10312.772,E2 -10312.772} C_VEL
LIN {X 0,Y 418.244,Z 700.38,A -85,B 0,C 180,E1 -10316.317,E2 -10316.317} C_VEL
LIN {X 0,Y 418.25,Z 700.382,A -85,B 0,C 180,E1 -10319.723,E2 -10319.723} C_VEL
LIN {X 0,Y 418.21,Z 700.39,A -85,B 0,C 180,E1 -10323.011,E2 -10323.011} C_VEL
LIN {X 0,Y 418.238,Z 700.385,A -85,B 0,C 180,E1 -10326.211,E2 -10326.211} C_VEL
LIN {X 0,Y 418.241,Z 700.39,A -85,B 0,C 180,E1 -10329.331,E2 -10329.331} C_VEL
LIN {X 0,Y 418.329,Z 700.551,A -85,B 0,C 180,E1 -10331.364,E2 -10331.364} C_VEL
LIN {X 0,Y 424.144,Z 715.929,A -85,B 0,C 180,E1 -10331.915,E2 -10331.915} C_VEL
LIN {X 0,Y 423.603,Z 781.501,A -85,B 0,C 180,E1 -10333.054,E2 -10333.054} C_VEL
LIN {X 0,Y 423.604,Z 794.297,A -85,B 0,C 180,E1 -10333.457,E2 -10333.457} C_VEL
LIN {X 0,Y 423.288,Z 806.693,A -85,B 0,C 180,E1 -10334.033,E2 -10334.033} C_VEL
LIN {X 0,Y 422.84,Z 817.903,A -85,B 0,C 180,E1 -10334.735,E2 -10334.735} C_VEL
LIN {X 0,Y 422.278,Z 829.376,A -85,B 0,C 180,E1 -10335.661,E2 -10335.661} C_VEL
LIN {X 0,Y 421.986,Z 834.739,A -85,B 0,C 180,E1 -10336.183,E2 -10336.183} C_VEL
LIN {X 0,Y 421.074,Z 839.485,A -85,B 0,C 180,E1 -10336.662,E2 -10336.662} C_VEL
LIN {X 0,Y 417.819,Z 846.966,A -85,B 0,C 180,E1 -10337.44,E2 -10337.44} C_VEL
LIN {X 0,Y 414.533,Z 853.894,A -85,B 0,C 180,E1 -10338.299,E2 -10338.299} C_VEL
LIN {X 0,Y 413.578,Z 857.738,A -85,B 0,C 180,E1 -10338.897,E2 -10338.897} C_VEL
LIN {X 0,Y 412.989,Z 864.606,A -85,B 0,C 180,E1 -10340.196,E2 -10340.196} C_VEL
LIN {X 0,Y 412.51,Z 870.284,A -85,B 0,C 180,E1 -10341.508,E2 -10341.508} C_VEL
LIN {X 0,Y 412.147,Z 875.904,A -85,B 0,C 180,E1 -10343.138,E2 -10343.138} C_VEL
LIN {X 0,Y 411.679,Z 879.799,A -85,B 0,C 180,E1 -10344.606,E2 -10344.606} C_VEL
LIN {X 0,Y 411.386,Z 882.666,A -85,B 0,C 180,E1 -10346.075,E2 -10346.075} C_VEL
LIN {X 0,Y 411.362,Z 884.028,A -85,B 0,C 180,E1 -10347.056,E2 -10347.056} C_VEL
LIN {X 0,Y 411.358,Z 884.993,A -85,B 0,C 180,E1 -10348.035,E2 -10348.035} C_VEL
LIN {X 0,Y 411.246,Z 885.836,A -85,B 0,C 180,E1 -10349.994,E2 -10349.994} C_VEL
LIN {X 0,Y 411.391,Z 885.077,A -85,B 0,C 180,E1 -10351.951,E2 -10351.951} C_VEL
LIN {X 0,Y 411.374,Z 882.846,A -85,B 0,C 180,E1 -10353.912,E2 -10353.912} C_VEL
LIN {X 0,Y 411.67,Z 880.038,A -85,B 0,C 180,E1 -10355.381,E2 -10355.381} C_VEL
LIN {X 0,Y 412.112,Z 876.22,A -85,B 0,C 180,E1 -10356.849,E2 -10356.849} C_VEL
LIN {X 0,Y 412.49,Z 870.749,A -85,B 0,C 180,E1 -10358.473,E2 -10358.473} C_VEL
LIN {X 0,Y 413.059,Z 863.942,A -85,B 0,C 180,E1 -10360.036,E2 -10360.036} C_VEL
LIN {X 0,Y 413.771,Z 855.925,A -85,B 0,C 180,E1 -10361.505,E2 -10361.505} C_VEL
LIN {X 0,Y 414.405,Z 847.71,A -85,B 0,C 180,E1 -10362.729,E2 -10362.729} C_VEL
LIN {X 0,Y 415.04,Z 837.554,A -85,B 0,C 180,E1 -10363.956,E2 -10363.956} C_VEL
LIN {X 0,Y 415.763,Z 827.099,A -85,B 0,C 180,E1 -10364.963,E2 -10364.963} C_VEL
LIN {X 0,Y 416.32,Z 815.324,A -85,B 0,C 180,E1 -10365.866,E2 -10365.866} C_VEL
LIN {X 0,Y 416.675,Z 802.818,A -85,B 0,C 180,E1 -10366.585,E2 -10366.585} C_VEL
LIN {X 0,Y 416.855,Z 789.714,A -85,B 0,C 180,E1 -10367.121,E2 -10367.121} C_VEL
LIN {X 0,Y 416.89,Z 777.269,A -85,B 0,C 180,E1 -10367.435,E2 -10367.435} C_VEL
LIN {X 0,Y 417.42,Z 717.352,A -85,B 0,C 180,E1 -10368.478,E2 -10368.478} C_VEL
LIN {X 0,Y 411.33,Z 701.565,A -85,B 0,C 180,E1 -10369.065,E2 -10369.065} C_VEL
LIN {X 0,Y 411.286,Z 701.257,A -85,B 0,C 180,E1 -10369.131,E2 -10369.131} C_VEL
LIN {X 0,Y 411.181,Z 701.263,A -85,B 0,C 180,E1 -10373.14,E2 -10373.14} C_VEL
LIN {X 0,Y 411.209,Z 701.256,A -85,B 0,C 180,E1 -10376.374,E2 -10376.374} C_VEL
LIN {X 0,Y 411.172,Z 701.265,A -85,B 0,C 180,E1 -10379.705,E2 -10379.705} C_VEL
LIN {X 0,Y 411.174,Z 701.269,A -85,B 0,C 180,E1 -10383.148,E2 -10383.148} C_VEL
LIN {X 0,Y 411.159,Z 701.266,A -85,B 0,C 180,E1 -10386.546,E2 -10386.546} C_VEL
LIN {X 0,Y 411.187,Z 701.264,A -85,B 0,C 180,E1 -10389.723,E2 -10389.723} C_VEL
LIN {X 0,Y 411.187,Z 701.266,A -85,B 0,C 180,E1 -10393.119,E2 -10393.119} C_VEL
LIN {X 0,Y 411.193,Z 701.254,A -85,B 0,C 180,E1 -10395.864,E2 -10395.864} C_VEL
LIN {X 0,Y 411.163,Z 701.271,A -85,B 0,C 180,E1 -10399.493,E2 -10399.493} C_VEL
LIN {X 0,Y 411.152,Z 701.271,A -85,B 0,C 180,E1 -10402.021,E2 -10402.021} C_VEL
LIN {X 0,Y 411.149,Z 701.268,A -85,B 0,C 180,E1 -10405.661,E2 -10405.661} C_VEL
LIN {X 0,Y 411.14,Z 701.267,A -85,B 0,C 180,E1 -10409.148,E2 -10409.148} C_VEL
LIN {X 0,Y 411.197,Z 701.264,A -85,B 0,C 180,E1 -10412.518,E2 -10412.518} C_VEL
LIN {X 0,Y 411.162,Z 701.264,A -85,B 0,C 180,E1 -10415.78,E2 -10415.78} C_VEL
LIN {X 0,Y 411.128,Z 701.271,A -85,B 0,C 180,E1 -10418.962,E2 -10418.962} C_VEL
LIN {X 0,Y 411.182,Z 701.262,A -85,B 0,C 180,E1 -10422.082,E2 -10422.082} C_VEL
LIN {X 0,Y 411.199,Z 701.262,A -85,B 0,C 180,E1 -10425.145,E2 -10425.145} C_VEL
LIN {X 0,Y 411.231,Z 701.257,A -85,B 0,C 180,E1 -10428.166,E2 -10428.166} C_VEL
LIN {X 0,Y 411.37,Z 701.242,A -85,B 0,C 180,E1 -10432.184,E2 -10432.184} C_VEL
LIN {X 0,Y 411.418,Z 701.235,A -85,B 0,C 180,E1 -10434.117,E2 -10434.117} C_VEL
LIN {X 0,Y 411.441,Z 701.231,A -85,B 0,C 180,E1 -10438.042,E2 -10438.042} C_VEL
LIN {X 0,Y 411.569,Z 701.217,A -85,B 0,C 180,E1 -10440,E2 -10440} C_VEL
LIN {X 0,Y 411.403,Z 701.234,A -85,B 0,C 180,E1 -10442.938,E2 -10442.938} C_VEL
LIN {X 0,Y 411.418,Z 701.236,A -85,B 0,C 180,E1 -10445.883,E2 -10445.883} C_VEL
LIN {X 0,Y 411.285,Z 701.25,A -85,B 0,C 180,E1 -10448.847,E2 -10448.847} C_VEL
LIN {X 0,Y 411.231,Z 701.26,A -85,B 0,C 180,E1 -10451.834,E2 -10451.834} C_VEL
LIN {X 0,Y 411.199,Z 701.262,A -85,B 0,C 180,E1 -10454.855,E2 -10454.855} C_VEL
LIN {X 0,Y 411.182,Z 701.266,A -85,B 0,C 180,E1 -10457.918,E2 -10457.918} C_VEL
LIN {X 0,Y 411.128,Z 701.264,A -85,B 0,C 180,E1 -10461.038,E2 -10461.038} C_VEL
LIN {X 0,Y 411.162,Z 701.265,A -85,B 0,C 180,E1 -10464.219,E2 -10464.219} C_VEL
LIN {X 0,Y 411.196,Z 701.261,A -85,B 0,C 180,E1 -10467.482,E2 -10467.482} C_VEL
LIN {X 0,Y 411.14,Z 701.264,A -85,B 0,C 180,E1 -10470.852,E2 -10470.852} C_VEL
LIN {X 0,Y 411.148,Z 701.269,A -85,B 0,C 180,E1 -10474.339,E2 -10474.339} C_VEL
LIN {X 0,Y 411.151,Z 701.262,A -85,B 0,C 180,E1 -10477.979,E2 -10477.979} C_VEL
LIN {X 0,Y 411.16,Z 701.267,A -85,B 0,C 180,E1 -10481.242,E2 -10481.242} C_VEL
LIN {X 0,Y 411.188,Z 701.266,A -85,B 0,C 180,E1 -10484.489,E2 -10484.489} C_VEL
LIN {X 0,Y 411.189,Z 701.258,A -85,B 0,C 180,E1 -10487.303,E2 -10487.303} C_VEL
LIN {X 0,Y 411.191,Z 701.262,A -85,B 0,C 180,E1 -10490.784,E2 -10490.784} C_VEL
LIN {X 0,Y 411.164,Z 701.272,A -85,B 0,C 180,E1 -10494.479,E2 -10494.479} C_VEL
LIN {X 0,Y 411.212,Z 701.417,A -85,B 0,C 180,E1 -10497.114,E2 -10497.114} C_VEL
LIN {X 0,Y 414.984,Z 717.563,A -85,B 0,C 180,E1 -10499.99,E2 -10499.99} C_VEL
LIN {X 0,Y 416.558,Z 725.41,A -85,B 0,C 180,E1 -10501.322,E2 -10501.322} C_VEL
LIN {X 0,Y 415.421,Z 742.395,A -85,B 0,C 180,E1 -10503.914,E2 -10503.914} C_VEL
LIN {X 0,Y 414.04,Z 764.707,A -85,B 0,C 180,E1 -10507.293,E2 -10507.293} C_VEL
LIN {X 0,Y 412.776,Z 786.508,A -85,B 0,C 180,E1 -10510.58,E2 -10510.58} C_VEL
LIN {X 0,Y 416.694,Z 822.643,A -85,B 0,C 180,E1 -10511.401,E2 -10511.401} C_VEL
LIN {X 0,Y 415.786,Z 897.247,A -85,B 0,C 180,E1 -10512.707,E2 -10512.707} C_VEL
LIN {X 0,Y 415.194,Z 911.228,A -85,B 0,C 180,E1 -10513.157,E2 -10513.157} C_VEL
LIN {X 0,Y 414.433,Z 923.767,A -85,B 0,C 180,E1 -10513.759,E2 -10513.759} C_VEL
LIN {X 0,Y 413.644,Z 934.987,A -85,B 0,C 180,E1 -10514.486,E2 -10514.486} C_VEL
LIN {X 0,Y 412.878,Z 945.386,A -85,B 0,C 180,E1 -10515.341,E2 -10515.341} C_VEL
LIN {X 0,Y 412.156,Z 955.765,A -85,B 0,C 180,E1 -10516.399,E2 -10516.399} C_VEL
LIN {X 0,Y 411.713,Z 964.164,A -85,B 0,C 180,E1 -10517.437,E2 -10517.437} C_VEL
LIN {X 0,Y 411.065,Z 974.016,A -85,B 0,C 180,E1 -10518.918,E2 -10518.918} C_VEL
LIN {X 0,Y 410.67,Z 981.9,A -85,B 0,C 180,E1 -10520.402,E2 -10520.402} C_VEL
LIN {X 0,Y 410.468,Z 989.2,A -85,B 0,C 180,E1 -10522.134,E2 -10522.134} C_VEL
LIN {X 0,Y 410.445,Z 994.118,A -85,B 0,C 180,E1 -10523.629,E2 -10523.629} C_VEL
LIN {X 0,Y 410.51,Z 997.829,A -85,B 0,C 180,E1 -10525.096,E2 -10525.096} C_VEL
LIN {X 0,Y 410.589,Z 999.767,A -85,B 0,C 180,E1 -10526.081,E2 -10526.081} C_VEL
LIN {X 0,Y 410.533,Z 1001.204,A -85,B 0,C 180,E1 -10527.063,E2 -10527.063} C_VEL
LIN {X 0,Y 410.551,Z 1002.236,A -85,B 0,C 180,E1 -10528.045,E2 -10528.045} C_VEL
LIN {X 0,Y 410.571,Z 1002.865,A -85,B 0,C 180,E1 -10529.026,E2 -10529.026} C_VEL
LIN {X 0,Y 410.591,Z 1003.088,A -85,B 0,C 180,E1 -10530.007,E2 -10530.007} C_VEL
LIN {X 0,Y 410.571,Z 1002.857,A -85,B 0,C 180,E1 -10530.987,E2 -10530.987} C_VEL
LIN {X 0,Y 410.552,Z 1002.221,A -85,B 0,C 180,E1 -10531.968,E2 -10531.968} C_VEL
LIN {X 0,Y 410.536,Z 1001.183,A -85,B 0,C 180,E1 -10532.95,E2 -10532.95} C_VEL
LIN {X 0,Y 410.593,Z 999.738,A -85,B 0,C 180,E1 -10533.932,E2 -10533.932} C_VEL
LIN {X 0,Y 410.436,Z 996.672,A -85,B 0,C 180,E1 -10535.41,E2 -10535.41} C_VEL
LIN {X 0,Y 410.428,Z 992.552,A -85,B 0,C 180,E1 -10536.89,E2 -10536.89} C_VEL
LIN {X 0,Y 410.552,Z 986.233,A -85,B 0,C 180,E1 -10538.621,E2 -10538.621} C_VEL
LIN {X 0,Y 410.754,Z 979.355,A -85,B 0,C 180,E1 -10540.107,E2 -10540.107} C_VEL
LIN {X 0,Y 411.259,Z 970.876,A -85,B 0,C 180,E1 -10541.589,E2 -10541.589} C_VEL
LIN {X 0,Y 411.887,Z 962.212,A -85,B 0,C 180,E1 -10542.822,E2 -10542.822} C_VEL
LIN {X 0,Y 412.248,Z 955.262,A -85,B 0,C 180,E1 -10543.654,E2 -10543.654} C_VEL
LIN {X 0,Y 412.89,Z 945.209,A -85,B 0,C 180,E1 -10544.672,E2 -10544.672} C_VEL
LIN {X 0,Y 413.665,Z 934.771,A -85,B 0,C 180,E1 -10545.526,E2 -10545.526} C_VEL
LIN {X 0,Y 414.523,Z 922.341,A -85,B 0,C 180,E1 -10546.314,E2 -10546.314} C_VEL
LIN {X 0,Y 415.296,Z 909.287,A -85,B 0,C 180,E1 -10546.915,E2 -10546.915} C_VEL
LIN {X 0,Y 415.793,Z 896.6,A -85,B 0,C 180,E1 -10547.306,E2 -10547.306} C_VEL
LIN {X 0,Y 416.598,Z 821.375,A -85,B 0,C 180,E1 -10548.621,E2 -10548.621} C_VEL
LIN {X 0,Y 413.685,Z 793.426,A -85,B 0,C 180,E1 -10549.281,E2 -10549.281} C_VEL
LIN {X 0,Y 412.816,Z 785.431,A -85,B 0,C 180,E1 -10549.556,E2 -10549.556} C_VEL
LIN {X 0,Y 414.209,Z 761.641,A -85,B 0,C 180,E1 -10553.167,E2 -10553.167} C_VEL
LIN {X 0,Y 415.567,Z 740.179,A -85,B 0,C 180,E1 -10556.414,E2 -10556.414} C_VEL
LIN {X 0,Y 416.52,Z 725.436,A -85,B 0,C 180,E1 -10558.669,E2 -10558.669} C_VEL
LIN {X 0,Y 413.808,Z 712.424,A -85,B 0,C 180,E1 -10560.9,E2 -10560.9} C_VEL
LIN {X 0,Y 411.18,Z 701.26,A -85,B 0,C 180,E1 -10562.936,E2 -10562.936} C_VEL
LIN {X 0,Y 411.186,Z 701.259,A -85,B 0,C 180,E1 -10566.748,E2 -10566.748} C_VEL
LIN {X 0,Y 411.179,Z 701.266,A -85,B 0,C 180,E1 -10569.722,E2 -10569.722} C_VEL
LIN {X 0,Y 411.136,Z 701.273,A -85,B 0,C 180,E1 -10573.144,E2 -10573.144} C_VEL
LIN {X 0,Y 411.178,Z 701.265,A -85,B 0,C 180,E1 -10575.885,E2 -10575.885} C_VEL
LIN {X 0,Y 411.164,Z 701.267,A -85,B 0,C 180,E1 -10578.777,E2 -10578.777} C_VEL
LIN {X 0,Y 411.199,Z 701.262,A -85,B 0,C 180,E1 -10582.027,E2 -10582.027} C_VEL
LIN {X 0,Y 411.219,Z 701.262,A -85,B 0,C 180,E1 -10585.126,E2 -10585.126} C_VEL
LIN {X 0,Y 411.182,Z 701.264,A -85,B 0,C 180,E1 -10588.004,E2 -10588.004} C_VEL
LIN {X 0,Y 411.196,Z 701.266,A -85,B 0,C 180,E1 -10591.408,E2 -10591.408} C_VEL
LIN {X 0,Y 411.235,Z 701.26,A -85,B 0,C 180,E1 -10594.934,E2 -10594.934} C_VEL
LIN {X 0,Y 411.221,Z 701.264,A -85,B 0,C 180,E1 -10597.914,E2 -10597.914} C_VEL
LIN {X 0,Y 411.306,Z 701.447,A -85,B 0,C 180,E1 -10600.52,E2 -10600.52} C_VEL
LIN {X 0,Y 412.404,Z 704.309,A -85,B 0,C 180,E1 -10600.681,E2 -10600.681} C_VEL
LIN {X 0,Y 418.061,Z 717.106,A -85,B 0,C 180,E1 -10601.399,E2 -10601.399} C_VEL
LIN {X 0,Y 416.88,Z 767.545,A -85,B 0,C 180,E1 -10602.556,E2 -10602.556} C_VEL
LIN {X 0,Y 416.651,Z 787.952,A -85,B 0,C 180,E1 -10603.052,E2 -10603.052} C_VEL
LIN {X 0,Y 416.592,Z 798.81,A -85,B 0,C 180,E1 -10603.46,E2 -10603.46} C_VEL
LIN {X 0,Y 416.343,Z 808.912,A -85,B 0,C 180,E1 -10603.967,E2 -10603.967} C_VEL
LIN {X 0,Y 415.98,Z 818.723,A -85,B 0,C 180,E1 -10604.593,E2 -10604.593} C_VEL
LIN {X 0,Y 415.622,Z 827.749,A -85,B 0,C 180,E1 -10605.307,E2 -10605.307} C_VEL
LIN {X 0,Y 415.124,Z 835.599,A -85,B 0,C 180,E1 -10606.04,E2 -10606.04} C_VEL
LIN {X 0,Y 414.647,Z 844.269,A -85,B 0,C 180,E1 -10607.022,E2 -10607.022} C_VEL
LIN {X 0,Y 414.142,Z 851.585,A -85,B 0,C 180,E1 -10608.002,E2 -10608.002} C_VEL
LIN {X 0,Y 413.68,Z 857.842,A -85,B 0,C 180,E1 -10608.981,E2 -10608.981} C_VEL
LIN {X 0,Y 413.202,Z 864.339,A -85,B 0,C 180,E1 -10610.207,E2 -10610.207} C_VEL
LIN {X 0,Y 412.774,Z 868.781,A -85,B 0,C 180,E1 -10611.185,E2 -10611.185} C_VEL
LIN {X 0,Y 412.416,Z 874.138,A -85,B 0,C 180,E1 -10612.657,E2 -10612.657} C_VEL
LIN {X 0,Y 411.823,Z 878.292,A -85,B 0,C 180,E1 -10614.123,E2 -10614.123} C_VEL
LIN {X 0,Y 411.726,Z 880.377,A -85,B 0,C 180,E1 -10615.104,E2 -10615.104} C_VEL
LIN {X 0,Y 411.488,Z 883.264,A -85,B 0,C 180,E1 -10617.063,E2 -10617.063} C_VEL
LIN {X 0,Y 411.25,Z 884.469,A -85,B 0,C 180,E1 -10619.021,E2 -10619.021} C_VEL
LIN {X 0,Y 411.197,Z 884.398,A -85,B 0,C 180,E1 -10620,E2 -10620} C_VEL
LIN {X 0,Y 411.201,Z 883.904,A -85,B 0,C 180,E1 -10620.979,E2 -10620.979} C_VEL
LIN {X 0,Y 411.028,Z 881.689,A -85,B 0,C 180,E1 -10622.94,E2 -10622.94} C_VEL
LIN {X 0,Y 411.24,Z 878.841,A -85,B 0,C 180,E1 -10624.411,E2 -10624.411} C_VEL
LIN {X 0,Y 411.491,Z 874.934,A -85,B 0,C 180,E1 -10625.882,E2 -10625.882} C_VEL
LIN {X 0,Y 411.805,Z 869.855,A -85,B 0,C 180,E1 -10627.354,E2 -10627.354} C_VEL
LIN {X 0,Y 412.005,Z 864.685,A -85,B 0,C 180,E1 -10628.579,E2 -10628.579} C_VEL
LIN {X 0,Y 412.327,Z 858.391,A -85,B 0,C 180,E1 -10629.814,E2 -10629.814} C_VEL
LIN {X 0,Y 412.73,Z 850.823,A -85,B 0,C 180,E1 -10631.044,E2 -10631.044} C_VEL
LIN {X 0,Y 413.107,Z 842.659,A -85,B 0,C 180,E1 -10632.154,E2 -10632.154} C_VEL
LIN {X 0,Y 413.477,Z 835.208,A -85,B 0,C 180,E1 -10633.016,E2 -10633.016} C_VEL
LIN {X 0,Y 413.895,Z 825.375,A -85,B 0,C 180,E1 -10633.964,E2 -10633.964} C_VEL
LIN {X 0,Y 414.253,Z 815.555,A -85,B 0,C 180,E1 -10634.743,E2 -10634.743} C_VEL
LIN {X 0,Y 414.554,Z 804.884,A -85,B 0,C 180,E1 -10635.424,E2 -10635.424} C_VEL
LIN {X 0,Y 414.809,Z 794.307,A -85,B 0,C 180,E1 -10635.95,E2 -10635.95} C_VEL
LIN {X 0,Y 415.018,Z 784.414,A -85,B 0,C 180,E1 -10636.32,E2 -10636.32} C_VEL
LIN {X 0,Y 415.081,Z 770.967,A -85,B 0,C 180,E1 -10636.665,E2 -10636.665} C_VEL
LIN {X 0,Y 415.792,Z 715.069,A -85,B 0,C 180,E1 -10637.799,E2 -10637.799} C_VEL
LIN {X 0,Y 411.267,Z 701.257,A -85,B 0,C 180,E1 -10638.268,E2 -10638.268} C_VEL
LIN {X 0,Y 411.213,Z 701.262,A -85,B 0,C 180,E1 -10641.033,E2 -10641.033} C_VEL
LIN {X 0,Y 411.22,Z 701.259,A -85,B 0,C 180,E1 -10644.216,E2 -10644.216} C_VEL
LIN {X 0,Y 411.199,Z 701.26,A -85,B 0,C 180,E1 -10647.482,E2 -10647.482} C_VEL
LIN {X 0,Y 411.216,Z 701.258,A -85,B 0,C 180,E1 -10649.712,E2 -10649.712} C_VEL
LIN {X 0,Y 411.223,Z 701.26,A -85,B 0,C 180,E1 -10653.154,E2 -10653.154} C_VEL
LIN {X 0,Y 411.21,Z 701.261,A -85,B 0,C 180,E1 -10656.55,E2 -10656.55} C_VEL
LIN {X 0,Y 411.187,Z 701.261,A -85,B 0,C 180,E1 -10659.718,E2 -10659.718} C_VEL
LIN {X 0,Y 411.181,Z 701.265,A -85,B 0,C 180,E1 -10663.133,E2 -10663.133} C_VEL
LIN {X 0,Y 411.182,Z 701.26,A -85,B 0,C 180,E1 -10665.879,E2 -10665.879} C_VEL
LIN {X 0,Y 411.176,Z 701.263,A -85,B 0,C 180,E1 -10669.49,E2 -10669.49} C_VEL
LIN {X 0,Y 411.198,Z 701.258,A -85,B 0,C 180,E1 -10672.022,E2 -10672.022} C_VEL
LIN {X 0,Y 411.217,Z 701.26,A -85,B 0,C 180,E1 -10675.121,E2 -10675.121} C_VEL
LIN {X 0,Y 411.17,Z 701.262,A -85,B 0,C 180,E1 -10677.998,E2 -10677.998} C_VEL
LIN {X 0,Y 411.183,Z 701.266,A -85,B 0,C 180,E1 -10681.402,E2 -10681.402} C_VEL
LIN {X 0,Y 411.202,Z 701.264,A -85,B 0,C 180,E1 -10684.937,E2 -10684.937} C_VEL
LIN {X 0,Y 411.21,Z 701.263,A -85,B 0,C 180,E1 -10687.908,E2 -10687.908} C_VEL
LIN {X 0,Y 411.269,Z 701.258,A -85,B 0,C 180,E1 -10691.016,E2 -10691.016} C_VEL
LIN {X 0,Y 413.381,Z 707.152,A -85,B 0,C 180,E1 -10691.238,E2 -10691.238} C_VEL
LIN {X 0,Y 417.434,Z 717.43,A -85,B 0,C 180,E1 -10691.622,E2 -10691.622} C_VEL
LIN {X 0,Y 416.867,Z 782.528,A -85,B 0,C 180,E1 -10692.772,E2 -10692.772} C_VEL
LIN {X 0,Y 416.861,Z 795.313,A -85,B 0,C 180,E1 -10693.182,E2 -10693.182} C_VEL
LIN {X 0,Y 416.533,Z 807.704,A -85,B 0,C 180,E1 -10693.767,E2 -10693.767} C_VEL
LIN {X 0,Y 416.069,Z 818.496,A -85,B 0,C 180,E1 -10694.449,E2 -10694.449} C_VEL
LIN {X 0,Y 415.537,Z 829.035,A -85,B 0,C 180,E1 -10695.298,E2 -10695.298} C_VEL
LIN {X 0,Y 414.87,Z 839.899,A -85,B 0,C 180,E1 -10696.4,E2 -10696.4} C_VEL
LIN {X 0,Y 414.323,Z 848.677,A -85,B 0,C 180,E1 -10697.504,E2 -10697.504} C_VEL
LIN {X 0,Y 413.578,Z 857.738,A -85,B 0,C 180,E1 -10698.897,E2 -10698.897} C_VEL
LIN {X 0,Y 412.648,Z 861.427,A -85,B 0,C 180,E1 -10699.522,E2 -10699.522} C_VEL
LIN {X 0,Y 409.44,Z 867.137,A -85,B 0,C 180,E1 -10700.557,E2 -10700.557} C_VEL
LIN {X 0,Y 406.26,Z 872.263,A -85,B 0,C 180,E1 -10701.663,E2 -10701.663} C_VEL
LIN {X 0,Y 405.386,Z 874.912,A -85,B 0,C 180,E1 -10702.393,E2 -10702.393} C_VEL
LIN {X 0,Y 405.106,Z 878.287,A -85,B 0,C 180,E1 -10703.519,E2 -10703.519} C_VEL
LIN {X 0,Y 404.557,Z 881.845,A -85,B 0,C 180,E1 -10705.011,E2 -10705.011} C_VEL
LIN {X 0,Y 404.374,Z 883.669,A -85,B 0,C 180,E1 -10706.007,E2 -10706.007} C_VEL
LIN {X 0,Y 404.345,Z 885.031,A -85,B 0,C 180,E1 -10707.005,E2 -10707.005} C_VEL
LIN {X 0,Y 404.343,Z 885.995,A -85,B 0,C 180,E1 -10708.001,E2 -10708.001} C_VEL
LIN {X 0,Y 404.222,Z 886.838,A -85,B 0,C 180,E1 -10709.993,E2 -10709.993} C_VEL
LIN {X 0,Y 404.37,Z 886.079,A -85,B 0,C 180,E1 -10711.985,E2 -10711.985} C_VEL
LIN {X 0,Y 404.362,Z 883.848,A -85,B 0,C 180,E1 -10713.98,E2 -10713.98} C_VEL
LIN {X 0,Y 404.674,Z 881.04,A -85,B 0,C 180,E1 -10715.474,E2 -10715.474} C_VEL
LIN {X 0,Y 405.139,Z 877.221,A -85,B 0,C 180,E1 -10716.967,E2 -10716.967} C_VEL
LIN {X 0,Y 405.54,Z 871.749,A -85,B 0,C 180,E1 -10718.619,E2 -10718.619} C_VEL
LIN {X 0,Y 406.141,Z 864.943,A -85,B 0,C 180,E1 -10720.209,E2 -10720.209} C_VEL
LIN {X 0,Y 406.892,Z 856.924,A -85,B 0,C 180,E1 -10721.702,E2 -10721.702} C_VEL
LIN {X 0,Y 407.552,Z 848.709,A -85,B 0,C 180,E1 -10722.947,E2 -10722.947} C_VEL
LIN {X 0,Y 408.223,Z 838.552,A -85,B 0,C 180,E1 -10724.194,E2 -10724.194} C_VEL
LIN {X 0,Y 408.973,Z 828.097,A -85,B 0,C 180,E1 -10725.217,E2 -10725.217} C_VEL
LIN {X 0,Y 409.535,Z 816.844,A -85,B 0,C 180,E1 -10726.098,E2 -10726.098} C_VEL
LIN {X 0,Y 409.941,Z 804.968,A -85,B 0,C 180,E1 -10726.808,E2 -10726.808} C_VEL
LIN {X 0,Y 410.128,Z 792.515,A -85,B 0,C 180,E1 -10727.346,E2 -10727.346} C_VEL
LIN {X 0,Y 410.208,Z 779.801,A -85,B 0,C 180,E1 -10727.696,E2 -10727.696} C_VEL
LIN {X 0,Y 410.718,Z 718.892,A -85,B 0,C 180,E1 -10728.781,E2 -10728.781} C_VEL
LIN {X 0,Y 404.268,Z 702.541,A -85,B 0,C 180,E1 -10729.413,E2 -10729.413} C_VEL
LIN {X 0,Y 404.208,Z 702.137,A -85,B 0,C 180,E1 -10729.45,E2 -10729.45} C_VEL
LIN {X 0,Y 404.134,Z 702.138,A -85,B 0,C 180,E1 -10732.826,E2 -10732.826} C_VEL
LIN {X 0,Y 404.157,Z 702.135,A -85,B 0,C 180,E1 -10735.759,E2 -10735.759} C_VEL
LIN {X 0,Y 404.169,Z 702.134,A -85,B 0,C 180,E1 -10737.992,E2 -10737.992} C_VEL
LIN {X 0,Y 404.109,Z 702.149,A -85,B 0,C 180,E1 -10741.55,E2 -10741.55} C_VEL
LIN {X 0,Y 404.151,Z 702.14,A -85,B 0,C 180,E1 -10745.009,E2 -10745.009} C_VEL
LIN {X 0,Y 404.124,Z 702.13,A -85,B 0,C 180,E1 -10748.749,E2 -10748.749} C_VEL
LIN {X 0,Y 404.149,Z 702.148,A -85,B 0,C 180,E1 -10751.604,E2 -10751.604} C_VEL
LIN {X 0,Y 404.156,Z 702.127,A -85,B 0,C 180,E1 -10754.523,E2 -10754.523} C_VEL
LIN {X 0,Y 404.162,Z 702.135,A -85,B 0,C 180,E1 -10757.299,E2 -10757.299} C_VEL
LIN {X 0,Y 404.119,Z 702.146,A -85,B 0,C 180,E1 -10759.949,E2 -10759.949} C_VEL
LIN {X 0,Y 404.086,Z 702.147,A -85,B 0,C 180,E1 -10763.118,E2 -10763.118} C_VEL
LIN {X 0,Y 404.088,Z 702.147,A -85,B 0,C 180,E1 -10766.182,E2 -10766.182} C_VEL
LIN {X 0,Y 404.094,Z 702.148,A -85,B 0,C 180,E1 -10769.71,E2 -10769.71} C_VEL
LIN {X 0,Y 404.132,Z 702.14,A -85,B 0,C 180,E1 -10773.118,E2 -10773.118} C_VEL
LIN {X 0,Y 404.112,Z 702.14,A -85,B 0,C 180,E1 -10775.33,E2 -10775.33} C_VEL
LIN {X 0,Y 404.092,Z 702.151,A -85,B 0,C 180,E1 -10778.578,E2 -10778.578} C_VEL
LIN {X 0,Y 404.14,Z 702.137,A -85,B 0,C 180,E1 -10781.759,E2 -10781.759} C_VEL
LIN {X 0,Y 404.144,Z 702.144,A -85,B 0,C 180,E1 -10784.88,E2 -10784.88} C_VEL
LIN {X 0,Y 404.201,Z 702.132,A -85,B 0,C 180,E1 -10787.957,E2 -10787.957} C_VEL
LIN {X 0,Y 404.311,Z 702.12,A -85,B 0,C 180,E1 -10792.006,E2 -10792.006} C_VEL
LIN {X 0,Y 404.364,Z 702.114,A -85,B 0,C 180,E1 -10794.014,E2 -10794.014} C_VEL
LIN {X 0,Y 404.411,Z 702.107,A -85,B 0,C 180,E1 -10798.008,E2 -10798.008} C_VEL
LIN {X 0,Y 404.539,Z 702.093,A -85,B 0,C 180,E1 -10800,E2 -10800} C_VEL
LIN {X 0,Y 404.36,Z 702.111,A -85,B 0,C 180,E1 -10802.989,E2 -10802.989} C_VEL
LIN {X 0,Y 404.364,Z 702.115,A -85,B 0,C 180,E1 -10805.986,E2 -10805.986} C_VEL
LIN {X 0,Y 404.224,Z 702.128,A -85,B 0,C 180,E1 -10809.002,E2 -10809.002} C_VEL
LIN {X 0,Y 404.201,Z 702.134,A -85,B 0,C 180,E1 -10812.043,E2 -10812.043} C_VEL
LIN {X 0,Y 404.144,Z 702.143,A -85,B 0,C 180,E1 -10815.12,E2 -10815.12} C_VEL
LIN {X 0,Y 404.14,Z 702.141,A -85,B 0,C 180,E1 -10818.241,E2 -10818.241} C_VEL
LIN {X 0,Y 404.071,Z 702.145,A -85,B 0,C 180,E1 -10821.423,E2 -10821.423} C_VEL
LIN {X 0,Y 404.112,Z 702.141,A -85,B 0,C 180,E1 -10824.67,E2 -10824.67} C_VEL
LIN {X 0,Y 404.135,Z 702.145,A -85,B 0,C 180,E1 -10828.004,E2 -10828.004} C_VEL
LIN {X 0,Y 404.087,Z 702.146,A -85,B 0,C 180,E1 -10831.565,E2 -10831.565} C_VEL
LIN {X 0,Y 404.128,Z 702.141,A -85,B 0,C 180,E1 -10835.022,E2 -10835.022} C_VEL
LIN {X 0,Y 404.112,Z 702.133,A -85,B 0,C 180,E1 -10838.762,E2 -10838.762} C_VEL
LIN {X 0,Y 404.141,Z 702.142,A -85,B 0,C 180,E1 -10841.617,E2 -10841.617} C_VEL
LIN {X 0,Y 404.153,Z 702.142,A -85,B 0,C 180,E1 -10844.537,E2 -10844.537} C_VEL
LIN {X 0,Y 404.167,Z 702.132,A -85,B 0,C 180,E1 -10847.312,E2 -10847.312} C_VEL
LIN {X 0,Y 404.128,Z 702.146,A -85,B 0,C 180,E1 -10849.963,E2 -10849.963} C_VEL
LIN {X 0,Y 404.103,Z 702.144,A -85,B 0,C 180,E1 -10853.132,E2 -10853.132} C_VEL
LIN {X 0,Y 404.111,Z 702.133,A -85,B 0,C 180,E1 -10856.195,E2 -10856.195} C_VEL
LIN {X 0,Y 404.146,Z 702.24,A -85,B 0,C 180,E1 -10856.768,E2 -10856.768} C_VEL
LIN {X 0,Y 407.988,Z 718.52,A -85,B 0,C 180,E1 -10859.734,E2 -10859.734} C_VEL
LIN {X 0,Y 409.584,Z 726.134,A -85,B 0,C 180,E1 -10861.057,E2 -10861.057} C_VEL
LIN {X 0,Y 409.45,Z 731.092,A -85,B 0,C 180,E1 -10861.844,E2 -10861.844} C_VEL
LIN {X 0,Y 407.835,Z 753.475,A -85,B 0,C 180,E1 -10865.308,E2 -10865.308} C_VEL
LIN {X 0,Y 406.431,Z 775.548,A -85,B 0,C 180,E1 -10868.716,E2 -10868.716} C_VEL
LIN {X 0,Y 405.804,Z 785.32,A -85,B 0,C 180,E1 -10870.23,E2 -10870.23} C_VEL
LIN {X 0,Y 409.957,Z 823.684,A -85,B 0,C 180,E1 -10871.12,E2 -10871.12} C_VEL
LIN {X 0,Y 409,Z 896.244,A -85,B 0,C 180,E1 -10872.411,E2 -10872.411} C_VEL
LIN {X 0,Y 408.389,Z 910.22,A -85,B 0,C 180,E1 -10872.868,E2 -10872.868} C_VEL
LIN {X 0,Y 407.597,Z 922.756,A -85,B 0,C 180,E1 -10873.479,E2 -10873.479} C_VEL
LIN {X 0,Y 406.779,Z 933.974,A -85,B 0,C 180,E1 -10874.218,E2 -10874.218} C_VEL
LIN {X 0,Y 405.857,Z 945.677,A -85,B 0,C 180,E1 -10875.21,E2 -10875.21} C_VEL
LIN {X 0,Y 405.095,Z 955.961,A -85,B 0,C 180,E1 -10876.3,E2 -10876.3} C_VEL
LIN {X 0,Y 404.766,Z 963.15,A -85,B 0,C 180,E1 -10877.218,E2 -10877.218} C_VEL
LIN {X 0,Y 404.117,Z 971.473,A -85,B 0,C 180,E1 -10878.471,E2 -10878.471} C_VEL
LIN {X 0,Y 403.667,Z 979.687,A -85,B 0,C 180,E1 -10879.981,E2 -10879.981} C_VEL
LIN {X 0,Y 403.467,Z 986.309,A -85,B 0,C 180,E1 -10881.493,E2 -10881.493} C_VEL
LIN {X 0,Y 403.41,Z 992.261,A -85,B 0,C 180,E1 -10883.23,E2 -10883.23} C_VEL
LIN {X 0,Y 403.445,Z 996.818,A -85,B 0,C 180,E1 -10885.01,E2 -10885.01} C_VEL
LIN {X 0,Y 403.552,Z 998.761,A -85,B 0,C 180,E1 -10886.012,E2 -10886.012} C_VEL
LIN {X 0,Y 403.493,Z 1000.198,A -85,B 0,C 180,E1 -10887.012,E2 -10887.012} C_VEL
LIN {X 0,Y 403.512,Z 1001.231,A -85,B 0,C 180,E1 -10888.011,E2 -10888.011} C_VEL
LIN {X 0,Y 403.538,Z 1001.862,A -85,B 0,C 180,E1 -10889.009,E2 -10889.009} C_VEL
LIN {X 0,Y 403.562,Z 1002.085,A -85,B 0,C 180,E1 -10890.007,E2 -10890.007} C_VEL
LIN {X 0,Y 403.538,Z 1001.853,A -85,B 0,C 180,E1 -10891.004,E2 -10891.004} C_VEL
LIN {X 0,Y 403.513,Z 1001.216,A -85,B 0,C 180,E1 -10892.003,E2 -10892.003} C_VEL
LIN {X 0,Y 403.496,Z 1000.177,A -85,B 0,C 180,E1 -10893.002,E2 -10893.002} C_VEL
LIN {X 0,Y 403.556,Z 998.731,A -85,B 0,C 180,E1 -10894.001,E2 -10894.001} C_VEL
LIN {X 0,Y 403.369,Z 995.658,A -85,B 0,C 180,E1 -10895.505,E2 -10895.505} C_VEL
LIN {X 0,Y 403.359,Z 991.535,A -85,B 0,C 180,E1 -10897.012,E2 -10897.012} C_VEL
LIN {X 0,Y 403.495,Z 985.213,A -85,B 0,C 180,E1 -10898.772,E2 -10898.772} C_VEL
LIN {X 0,Y 403.704,Z 978.331,A -85,B 0,C 180,E1 -10900.285,E2 -10900.285} C_VEL
LIN {X 0,Y 404.236,Z 969.851,A -85,B 0,C 180,E1 -10901.794,E2 -10901.794} C_VEL
LIN {X 0,Y 404.894,Z 961.186,A -85,B 0,C 180,E1 -10903.047,E2 -10903.047} C_VEL
LIN {X 0,Y 405.332,Z 954.174,A -85,B 0,C 180,E1 -10903.9,E2 -10903.9} C_VEL
LIN {X 0,Y 405.92,Z 944.178,A -85,B 0,C 180,E1 -10904.93,E2 -10904.93} C_VEL
LIN {X 0,Y 406.798,Z 933.749,A -85,B 0,C 180,E1 -10905.795,E2 -10905.795} C_VEL
LIN {X 0,Y 407.623,Z 922.455,A -85,B 0,C 180,E1 -10906.534,E2 -10906.534} C_VEL
LIN {X 0,Y 408.399,Z 909.793,A -85,B 0,C 180,E1 -10907.145,E2 -10907.145} C_VEL
LIN {X 0,Y 408.977,Z 896.733,A -85,B 0,C 180,E1 -10907.571,E2 -10907.571} C_VEL
LIN {X 0,Y 409.915,Z 822.843,A -85,B 0,C 180,E1 -10908.891,E2 -10908.891} C_VEL
LIN {X 0,Y 407.999,Z 804.052,A -85,B 0,C 180,E1 -10909.359,E2 -10909.359} C_VEL
LIN {X 0,Y 406.262,Z 786.642,A -85,B 0,C 180,E1 -10909.921,E2 -10909.921} C_VEL
LIN {X 0,Y 405.904,Z 783.56,A -85,B 0,C 180,E1 -10910.035,E2 -10910.035} C_VEL
LIN {X 0,Y 407.529,Z 758.341,A -85,B 0,C 180,E1 -10913.935,E2 -10913.935} C_VEL
LIN {X 0,Y 409.181,Z 734.386,A -85,B 0,C 180,E1 -10917.634,E2 -10917.634} C_VEL
LIN {X 0,Y 409.696,Z 727.487,A -85,B 0,C 180,E1 -10918.711,E2 -10918.711} C_VEL
LIN {X 0,Y 407.337,Z 715.816,A -85,B 0,C 180,E1 -10920.741,E2 -10920.741} C_VEL
LIN {X 0,Y 404.101,Z 702.145,A -85,B 0,C 180,E1 -10923.275,E2 -10923.275} C_VEL
LIN {X 0,Y 404.133,Z 702.138,A -85,B 0,C 180,E1 -10926.874,E2 -10926.874} C_VEL
LIN {X 0,Y 404.135,Z 702.142,A -85,B 0,C 180,E1 -10930.078,E2 -10930.078} C_VEL
LIN {X 0,Y 404.094,Z 702.149,A -85,B 0,C 180,E1 -10933.075,E2 -10933.075} C_VEL
LIN {X 0,Y 404.135,Z 702.142,A -85,B 0,C 180,E1 -10935.924,E2 -10935.924} C_VEL
LIN {X 0,Y 404.119,Z 702.144,A -85,B 0,C 180,E1 -10938.635,E2 -10938.635} C_VEL
LIN {X 0,Y 404.155,Z 702.144,A -85,B 0,C 180,E1 -10941.498,E2 -10941.498} C_VEL
LIN {X 0,Y 404.19,Z 702.136,A -85,B 0,C 180,E1 -10944.984,E2 -10944.984} C_VEL
LIN {X 0,Y 404.156,Z 702.139,A -85,B 0,C 180,E1 -10948.444,E2 -10948.444} C_VEL
LIN {X 0,Y 404.17,Z 702.141,A -85,B 0,C 180,E1 -10950.864,E2 -10950.864} C_VEL
LIN {X 0,Y 404.159,Z 702.141,A -85,B 0,C 180,E1 -10954.232,E2 -10954.232} C_VEL
LIN {X 0,Y 404.185,Z 702.139,A -85,B 0,C 180,E1 -10957.509,E2 -10957.509} C_VEL
LIN {X 0,Y 404.209,Z 702.138,A -85,B 0,C 180,E1 -10959.993,E2 -10959.993} C_VEL
LIN {X 0,Y 405.212,Z 704.97,A -85,B 0,C 180,E1 -10960.154,E2 -10960.154} C_VEL
LIN {X 0,Y 410.358,Z 715.937,A -85,B 0,C 180,E1 -10960.846,E2 -10960.846} C_VEL
LIN {X 0,Y 411.76,Z 719.571,A -85,B 0,C 180,E1 -10961.042,E2 -10961.042} C_VEL
LIN {X 0,Y 410.137,Z 784.025,A -85,B 0,C 180,E1 -10962.55,E2 -10962.55} C_VEL
LIN {X 0,Y 410.075,Z 797.905,A -85,B 0,C 180,E1 -10963.029,E2 -10963.029} C_VEL
LIN {X 0,Y 409.771,Z 809.568,A -85,B 0,C 180,E1 -10963.612,E2 -10963.612} C_VEL
LIN {X 0,Y 409.39,Z 819.393,A -85,B 0,C 180,E1 -10964.241,E2 -10964.241} C_VEL
LIN {X 0,Y 409.03,Z 827.837,A -85,B 0,C 180,E1 -10964.903,E2 -10964.903} C_VEL
LIN {X 0,Y 408.405,Z 837.347,A -85,B 0,C 180,E1 -10965.805,E2 -10965.805} C_VEL
LIN {X 0,Y 407.937,Z 845.933,A -85,B 0,C 180,E1 -10966.805,E2 -10966.805} C_VEL
LIN {X 0,Y 407.361,Z 853.174,A -85,B 0,C 180,E1 -10967.799,E2 -10967.799} C_VEL
LIN {X 0,Y 406.864,Z 859.343,A -85,B 0,C 180,E1 -10968.795,E2 -10968.795} C_VEL
LIN {X 0,Y 406.345,Z 865.759,A -85,B 0,C 180,E1 -10970.04,E2 -10970.04} C_VEL
LIN {X 0,Y 405.918,Z 870.16,A -85,B 0,C 180,E1 -10971.035,E2 -10971.035} C_VEL
LIN {X 0,Y 405.517,Z 875.461,A -85,B 0,C 180,E1 -10972.531,E2 -10972.531} C_VEL
LIN {X 0,Y 404.877,Z 879.572,A -85,B 0,C 180,E1 -10974.022,E2 -10974.022} C_VEL
LIN {X 0,Y 404.769,Z 881.654,A -85,B 0,C 180,E1 -10975.02,E2 -10975.02} C_VEL
LIN {X 0,Y 404.498,Z 884.45,A -85,B 0,C 180,E1 -10977.012,E2 -10977.012} C_VEL
LIN {X 0,Y 404.31,Z 885.232,A -85,B 0,C 180,E1 -10978.008,E2 -10978.008} C_VEL
LIN {X 0,Y 404.241,Z 885.589,A -85,B 0,C 180,E1 -10979.004,E2 -10979.004} C_VEL
LIN {X 0,Y 404.179,Z 885.469,A -85,B 0,C 180,E1 -10980,E2 -10980} C_VEL
LIN {X 0,Y 404.182,Z 884.941,A -85,B 0,C 180,E1 -10980.996,E2 -10980.996} C_VEL
LIN {X 0,Y 403.999,Z 882.62,A -85,B 0,C 180,E1 -10982.992,E2 -10982.992} C_VEL
LIN {X 0,Y 404.225,Z 879.702,A -85,B 0,C 180,E1 -10984.487,E2 -10984.487} C_VEL
LIN {X 0,Y 404.495,Z 875.716,A -85,B 0,C 180,E1 -10985.984,E2 -10985.984} C_VEL
LIN {X 0,Y 404.816,Z 870.548,A -85,B 0,C 180,E1 -10987.482,E2 -10987.482} C_VEL
LIN {X 0,Y 405.016,Z 865.437,A -85,B 0,C 180,E1 -10988.698,E2 -10988.698} C_VEL
LIN {X 0,Y 405.365,Z 858.89,A -85,B 0,C 180,E1 -10989.984,E2 -10989.984} C_VEL
LIN {X 0,Y 405.765,Z 851.198,A -85,B 0,C 180,E1 -10991.236,E2 -10991.236} C_VEL
LIN {X 0,Y 406.111,Z 843.919,A -85,B 0,C 180,E1 -10992.239,E2 -10992.239} C_VEL
LIN {X 0,Y 406.561,Z 835.286,A -85,B 0,C 180,E1 -10993.241,E2 -10993.241} C_VEL
LIN {X 0,Y 406.938,Z 826.594,A -85,B 0,C 180,E1 -10994.091,E2 -10994.091} C_VEL
LIN {X 0,Y 407.308,Z 816.376,A -85,B 0,C 180,E1 -10994.914,E2 -10994.914} C_VEL
LIN {X 0,Y 407.621,Z 806.399,A -85,B 0,C 180,E1 -10995.564,E2 -10995.564} C_VEL
LIN {X 0,Y 407.836,Z 795.991,A -85,B 0,C 180,E1 -10996.101,E2 -10996.101} C_VEL
LIN {X 0,Y 408.092,Z 785.379,A -85,B 0,C 180,E1 -10996.509,E2 -10996.509} C_VEL
LIN {X 0,Y 408.166,Z 773.576,A -85,B 0,C 180,E1 -10996.827,E2 -10996.827} C_VEL
LIN {X 0,Y 408.934,Z 716.534,A -85,B 0,C 180,E1 -10998.014,E2 -10998.014} C_VEL
LIN {X 0,Y 404.224,Z 702.135,A -85,B 0,C 180,E1 -10998.533,E2 -10998.533} C_VEL
LIN {X 0,Y 404.155,Z 702.138,A -85,B 0,C 180,E1 -11001.419,E2 -11001.419} C_VEL
LIN {X 0,Y 404.174,Z 702.141,A -85,B 0,C 180,E1 -11004.666,E2 -11004.666} C_VEL
LIN {X 0,Y 404.141,Z 702.138,A -85,B 0,C 180,E1 -11008.004,E2 -11008.004} C_VEL
LIN {X 0,Y 404.163,Z 702.138,A -85,B 0,C 180,E1 -11010.284,E2 -11010.284} C_VEL
LIN {X 0,Y 404.156,Z 702.136,A -85,B 0,C 180,E1 -11013.811,E2 -11013.811} C_VEL
LIN {X 0,Y 404.153,Z 702.142,A -85,B 0,C 180,E1 -11016.872,E2 -11016.872} C_VEL
LIN {X 0,Y 404.136,Z 702.139,A -85,B 0,C 180,E1 -11020.073,E2 -11020.073} C_VEL
LIN {X 0,Y 404.161,Z 702.14,A -85,B 0,C 180,E1 -11023.079,E2 -11023.079} C_VEL
LIN {X 0,Y 404.138,Z 702.137,A -85,B 0,C 180,E1 -11025.919,E2 -11025.919} C_VEL
LIN {X 0,Y 404.119,Z 702.142,A -85,B 0,C 180,E1 -11028.63,E2 -11028.63} C_VEL
LIN {X 0,Y 404.155,Z 702.138,A -85,B 0,C 180,E1 -11031.492,E2 -11031.492} C_VEL
LIN {X 0,Y 404.188,Z 702.135,A -85,B 0,C 180,E1 -11034.979,E2 -11034.979} C_VEL
LIN {X 0,Y 404.147,Z 702.137,A -85,B 0,C 180,E1 -11038.441,E2 -11038.441} C_VEL
LIN {X 0,Y 404.163,Z 702.138,A -85,B 0,C 180,E1 -11040.858,E2 -11040.858} C_VEL
LIN {X 0,Y 404.166,Z 702.138,A -85,B 0,C 180,E1 -11044.719,E2 -11044.719} C_VEL
LIN {X 0,Y 404.177,Z 702.141,A -85,B 0,C 180,E1 -11047.503,E2 -11047.503} C_VEL
LIN {X 0,Y 404.208,Z 702.136,A -85,B 0,C 180,E1 -11050.663,E2 -11050.663} C_VEL
LIN {X 0,Y 406.399,Z 708.061,A -85,B 0,C 180,E1 -11050.9,E2 -11050.9} C_VEL
LIN {X 0,Y 410.732,Z 719.091,A -85,B 0,C 180,E1 -11051.322,E2 -11051.322} C_VEL
LIN {X 0,Y 410.142,Z 782.064,A -85,B 0,C 180,E1 -11052.448,E2 -11052.448} C_VEL
LIN {X 0,Y 410.152,Z 794.774,A -85,B 0,C 180,E1 -11052.834,E2 -11052.834} C_VEL
LIN {X 0,Y 409.845,Z 807.596,A -85,B 0,C 180,E1 -11053.431,E2 -11053.431} C_VEL
LIN {X 0,Y 409.303,Z 819.502,A -85,B 0,C 180,E1 -11054.186,E2 -11054.186} C_VEL
LIN {X 0,Y 408.743,Z 830.043,A -85,B 0,C 180,E1 -11055.048,E2 -11055.048} C_VEL
LIN {X 0,Y 408.043,Z 840.906,A -85,B 0,C 180,E1 -11056.168,E2 -11056.168} C_VEL
LIN {X 0,Y 407.465,Z 849.683,A -85,B 0,C 180,E1 -11057.29,E2 -11057.29} C_VEL
LIN {X 0,Y 406.684,Z 858.773,A -85,B 0,C 180,E1 -11058.711,E2 -11058.711} C_VEL
LIN {X 0,Y 406.066,Z 865.611,A -85,B 0,C 180,E1 -11060.027,E2 -11060.027} C_VEL
LIN {X 0,Y 405.561,Z 871.287,A -85,B 0,C 180,E1 -11061.361,E2 -11061.361} C_VEL
LIN {X 0,Y 405.386,Z 874.912,A -85,B 0,C 180,E1 -11062.393,E2 -11062.393} C_VEL
LIN {X 0,Y 404.559,Z 876.649,A -85,B 0,C 180,E1 -11062.888,E2 -11062.888} C_VEL
LIN {X 0,Y 401.464,Z 879.398,A -85,B 0,C 180,E1 -11063.648,E2 -11063.648} C_VEL
LIN {X 0,Y 398.364,Z 881.781,A -85,B 0,C 180,E1 -11064.439,E2 -11064.439} C_VEL
LIN {X 0,Y 397.543,Z 882.945,A -85,B 0,C 180,E1 -11064.976,E2 -11064.976} C_VEL
LIN {X 0,Y 397.363,Z 884.673,A -85,B 0,C 180,E1 -11065.937,E2 -11065.937} C_VEL
LIN {X 0,Y 397.328,Z 886.034,A -85,B 0,C 180,E1 -11066.952,E2 -11066.952} C_VEL
LIN {X 0,Y 397.326,Z 886.997,A -85,B 0,C 180,E1 -11067.966,E2 -11067.966} C_VEL
LIN {X 0,Y 397.197,Z 887.84,A -85,B 0,C 180,E1 -11069.993,E2 -11069.993} C_VEL
LIN {X 0,Y 397.35,Z 887.081,A -85,B 0,C 180,E1 -11072.02,E2 -11072.02} C_VEL
LIN {X 0,Y 397.35,Z 884.85,A -85,B 0,C 180,E1 -11074.05,E2 -11074.05} C_VEL
LIN {X 0,Y 397.68,Z 882.041,A -85,B 0,C 180,E1 -11075.571,E2 -11075.571} C_VEL
LIN {X 0,Y 398.169,Z 878.222,A -85,B 0,C 180,E1 -11077.09,E2 -11077.09} C_VEL
LIN {X 0,Y 398.592,Z 872.75,A -85,B 0,C 180,E1 -11078.771,E2 -11078.771} C_VEL
LIN {X 0,Y 399.226,Z 865.943,A -85,B 0,C 180,E1 -11080.388,E2 -11080.388} C_VEL
LIN {X 0,Y 400.017,Z 857.923,A -85,B 0,C 180,E1 -11081.906,E2 -11081.906} C_VEL
LIN {X 0,Y 400.706,Z 849.709,A -85,B 0,C 180,E1 -11083.172,E2 -11083.172} C_VEL
LIN {X 0,Y 401.414,Z 839.551,A -85,B 0,C 180,E1 -11084.439,E2 -11084.439} C_VEL
LIN {X 0,Y 402.2,Z 829.096,A -85,B 0,C 180,E1 -11085.48,E2 -11085.48} C_VEL
LIN {X 0,Y 402.787,Z 817.84,A -85,B 0,C 180,E1 -11086.375,E2 -11086.375} C_VEL
LIN {X 0,Y 403.211,Z 805.962,A -85,B 0,C 180,E1 -11087.097,E2 -11087.097} C_VEL
LIN {X 0,Y 403.414,Z 792.601,A -85,B 0,C 180,E1 -11087.677,E2 -11087.677} C_VEL
LIN {X 0,Y 403.486,Z 779.224,A -85,B 0,C 180,E1 -11088.034,E2 -11088.034} C_VEL
LIN {X 0,Y 404.016,Z 720.529,A -85,B 0,C 180,E1 -11089.092,E2 -11089.092} C_VEL
LIN {X 0,Y 397.179,Z 703.259,A -85,B 0,C 180,E1 -11089.78,E2 -11089.78} C_VEL
LIN {X 0,Y 397.154,Z 703.015,A -85,B 0,C 180,E1 -11089.908,E2 -11089.908} C_VEL
LIN {X 0,Y 397.107,Z 703.014,A -85,B 0,C 180,E1 -11094.011,E2 -11094.011} C_VEL
LIN {X 0,Y 397.168,Z 703.009,A -85,B 0,C 180,E1 -11097.382,E2 -11097.382} C_VEL
LIN {X 0,Y 397.049,Z 703.025,A -85,B 0,C 180,E1 -11100.875,E2 -11100.875} C_VEL
LIN {X 0,Y 397.092,Z 703.017,A -85,B 0,C 180,E1 -11104.486,E2 -11104.486} C_VEL
LIN {X 0,Y 397.071,Z 703.008,A -85,B 0,C 180,E1 -11108.267,E2 -11108.267} C_VEL
LIN {X 0,Y 397.114,Z 703.02,A -85,B 0,C 180,E1 -11111.986,E2 -11111.986} C_VEL
LIN {X 0,Y 397.106,Z 703.004,A -85,B 0,C 180,E1 -11115.053,E2 -11115.053} C_VEL
LIN {X 0,Y 397.108,Z 703.023,A -85,B 0,C 180,E1 -11118,E2 -11118} C_VEL
LIN {X 0,Y 397.058,Z 703.023,A -85,B 0,C 180,E1 -11121.72,E2 -11121.72} C_VEL
LIN {X 0,Y 397.069,Z 703.021,A -85,B 0,C 180,E1 -11125.501,E2 -11125.501} C_VEL
LIN {X 0,Y 397.027,Z 703.025,A -85,B 0,C 180,E1 -11129.113,E2 -11129.113} C_VEL
LIN {X 0,Y 397.132,Z 703.015,A -85,B 0,C 180,E1 -11132.605,E2 -11132.605} C_VEL
LIN {X 0,Y 397.068,Z 703.021,A -85,B 0,C 180,E1 -11135.977,E2 -11135.977} C_VEL
LIN {X 0,Y 397.071,Z 703.021,A -85,B 0,C 180,E1 -11139.701,E2 -11139.701} C_VEL
LIN {X 0,Y 397.114,Z 703.011,A -85,B 0,C 180,E1 -11142.841,E2 -11142.841} C_VEL
LIN {X 0,Y 397.114,Z 703.016,A -85,B 0,C 180,E1 -11145.654,E2 -11145.654} C_VEL
LIN {X 0,Y 397.141,Z 703.008,A -85,B 0,C 180,E1 -11148.775,E2 -11148.775} C_VEL
LIN {X 0,Y 397.29,Z 702.995,A -85,B 0,C 180,E1 -11152.073,E2 -11152.073} C_VEL
LIN {X 0,Y 397.192,Z 703.005,A -85,B 0,C 180,E1 -11154.924,E2 -11154.924} C_VEL
LIN {X 0,Y 397.38,Z 702.983,A -85,B 0,C 180,E1 -11157.973,E2 -11157.973} C_VEL
LIN {X 0,Y 397.509,Z 702.969,A -85,B 0,C 180,E1 -11160,E2 -11160} C_VEL
LIN {X 0,Y 397.318,Z 702.988,A -85,B 0,C 180,E1 -11163.042,E2 -11163.042} C_VEL
LIN {X 0,Y 397.313,Z 702.993,A -85,B 0,C 180,E1 -11166.092,E2 -11166.092} C_VEL
LIN {X 0,Y 397.186,Z 703.004,A -85,B 0,C 180,E1 -11169.163,E2 -11169.163} C_VEL
LIN {X 0,Y 397.16,Z 703.011,A -85,B 0,C 180,E1 -11172.26,E2 -11172.26} C_VEL
LIN {X 0,Y 397.116,Z 703.022,A -85,B 0,C 180,E1 -11175.395,E2 -11175.395} C_VEL
LIN {X 0,Y 397.092,Z 703.018,A -85,B 0,C 180,E1 -11178.577,E2 -11178.577} C_VEL
LIN {X 0,Y 397.029,Z 703.026,A -85,B 0,C 180,E1 -11181.822,E2 -11181.822} C_VEL
LIN {X 0,Y 397.092,Z 703.017,A -85,B 0,C 180,E1 -11185.136,E2 -11185.136} C_VEL
LIN {X 0,Y 397.101,Z 703.021,A -85,B 0,C 180,E1 -11187.781,E2 -11187.781} C_VEL
LIN {X 0,Y 397.026,Z 703.022,A -85,B 0,C 180,E1 -11190.887,E2 -11190.887} C_VEL
LIN {X 0,Y 397.068,Z 703.022,A -85,B 0,C 180,E1 -11194.499,E2 -11194.499} C_VEL
LIN {X 0,Y 397.057,Z 703.014,A -85,B 0,C 180,E1 -11198.28,E2 -11198.28} C_VEL
LIN {X 0,Y 397.106,Z 703.022,A -85,B 0,C 180,E1 -11202,E2 -11202} C_VEL
LIN {X 0,Y 397.105,Z 703.018,A -85,B 0,C 180,E1 -11205.066,E2 -11205.066} C_VEL
LIN {X 0,Y 397.114,Z 703.012,A -85,B 0,C 180,E1 -11208.014,E2 -11208.014} C_VEL
LIN {X 0,Y 397.071,Z 703.023,A -85,B 0,C 180,E1 -11211.733,E2 -11211.733} C_VEL
LIN {X 0,Y 397.091,Z 703.012,A -85,B 0,C 180,E1 -11215.514,E2 -11215.514} C_VEL
LIN {X 0,Y 397.11,Z 703.09,A -85,B 0,C 180,E1 -11216.416,E2 -11216.416} C_VEL
LIN {X 0,Y 400.999,Z 719.431,A -85,B 0,C 180,E1 -11219.462,E2 -11219.462} C_VEL
LIN {X 0,Y 402.757,Z 728.047,A -85,B 0,C 180,E1 -11220.989,E2 -11220.989} C_VEL
LIN {X 0,Y 401.789,Z 742.326,A -85,B 0,C 180,E1 -11223.257,E2 -11223.257} C_VEL
LIN {X 0,Y 400.069,Z 766.111,A -85,B 0,C 180,E1 -11227.001,E2 -11227.001} C_VEL
